// TwinCAT 3 PLC project ProgrammHalle
// ProgramVersion: 3.1.4022.1
// libraries:
//   OSCAT, * (RWTH Aachen University - E.ON Energy Research Center)
//   Tc2_ModbusRTU, * (Beckhoff Automation GmbH)
//   Tc2_Standard, * (Beckhoff Automation GmbH)
//   Tc2_System, * (Beckhoff Automation GmbH)
//   Tc3_BA2_Common, * (Beckhoff Automation GmbH)
//   Tc3_BACnetRev14, * (Beckhoff Automation GmbH)
//   Tc3_BA_Common, * (Beckhoff Automation GmbH)
//   Tc3_IotBase, * (Beckhoff Automation GmbH)
//   Tc3_Module, * (Beckhoff Automation GmbH)
//   TcUnit, * (www.tcunit.org)
// project tree:
//   DUTs/ E_ControlMode.TcDUT, E_PumpControlMode.TcDUT
//   GVLs/ ADS.TcGVL, GVL.TcGVL
//   / PlcTask.TcTTO
//   POUs/Components/ FB_ExhAirModbus.TcPOU, FB_FanBACnet.TcPOU, FB_FanControl.TcPOU, FB_HydMixCir.TcPOU, FB_HydThrotCir.TcPOU, FB_JetNozzle1.TcPOU, FB_JetNozzle2.TcPOU, FB_PumpBACnet.TcPOU, FB_PumpBACnet1.TcPOU, FB_PumpBACnet2.TcPOU, FB_PumpWiloIF.TcPOU, FB_RoomControlUnit.TcPOU, FB_SenTempEL321x.TcPOU, FB_TempSensPt100.TcPOU, FB_TVJModbusMaster.TcPOU, FB_TVRModbusMaster.TcPOU, FB_ValveBACnet.TcPOU, FB_Valve_0_10V.TcPOU, FB_Valve_2_10V.TcPOU, FB_Valve_4_20A.TcPOU, FB_VFCModbus1.TcPOU, FB_VFCModbus2.TcPOU, FB_VVS_JN.TcPOU, FC_CoolingCurve.TcPOU, FC_Current4_20Raw_TO_Percentage.TcPOU, FC_HeatingCurve.TcPOU, FC_MeanOfArray.TcPOU, FC_Percentage_TO_Current4_20Raw.TcPOU, FC_Percentage_TO_Voltage0_10Raw.TcPOU, FC_Percentage_TO_Voltage2_10Raw.TcPOU, FC_Pt100Raw_TO_Temperature.TcPOU, FC_Voltage0_10Raw_TO_Percentage.TcPOU, FC_Voltage2_10Raw_TO_Percentage.TcPOU
//   POUs/EnvTemperature/ FB_AmbientAir.TcPOU
//   POUs/HeatSupplySystem/ FB_HSS.TcPOU, FB_HSSController.TcPOU
//   POUs/Interfaces/ I_Controller.TcIO, I_HydraulicMixingControl.TcIO, I_HydraulicThrottlingControl.TcIO, I_JetNozzle.TcIO, I_Pump.TcIO, I_TemperatureSensor.TcIO, I_Valve.TcIO, I_VolumeFlowController.TcIO
//   POUs/ MAIN.TcPOU
//   POUs/SensorData/ FB_SenDaHydMixCir.TcPOU
//   POUs/Test/Components_Test/ FC_HeatingCurve_Test.TcPOU
//   POUs/Test/HeatSupplySystem_Test/ FB_HSSController_Test.TcPOU
//   POUs/Test/ PRG_TEST.TcPOU

CONFIGURATION ProgrammHalle
    RESOURCE PLC ON TwinCAT3
        TASK PlcTask(INTERVAL := T#10ms, PRIORITY := 20);
        PROGRAM MAIN WITH PlcTask : MAIN;
        PROGRAM PRG_TEST WITH PlcTask : PRG_TEST;
    END_RESOURCE
END_CONFIGURATION

// ---- DUTs/E_ControlMode.TcDUT
{attribute 'qualified_only'}
{attribute 'strict'}
TYPE E_ControlMode :
(
	Off, 				(*0*)
	Init, 				(*1*)
	OperationTest, 		(*2*)
	Auto, 				(*3*)
	Manual,				(*4*)
	ExternalADSControl	(*5*)
);
END_TYPE

// ---- DUTs/E_PumpControlMode.TcDUT
{attribute 'qualified_only'}
{attribute 'strict'}
TYPE E_PumpControlMode :
(
	OFF := 0,					
	CONST_SPEED := 1,				
	CONST_DIFFPRESS := 6,		
	VAR_DIFFPRESS := 7,
	NONE := 99
);
END_TYPE

// ---- GVLs/ADS.TcGVL
{attribute 'qualified_only'}
VAR_GLOBAL
	
	//Modes
	eModeMainControlModeADS	AT %I*	: E_ControlMode := E_ControlMode.Auto; //W
	
	eModeHSSADS			AT %I*	: E_ControlMode := E_ControlMode.Auto; //W
	

	//Ambient air datapoints
	fTempAmbAirADS				AT %Q* 	: REAL;
	fTemperatureAmbientMeanADS 	AT %Q*	: REAL;

	
	//HSS  datapoints
	//Temperature sensor datapoints
	fHSSTempSupPrimADS 	AT %Q*	: REAL;
	fHSSTempRetPrimADS 	AT %Q*	: REAL;
	fHSSTempSupADS 		AT %Q*	: REAL;
	fHSSTempRetADS 		AT %Q*	: REAL;
	//Valve datapoints
	fHSSValveActADS 		AT %Q*	: REAL;
	fHSSValveSetADS 		AT %I*	: REAL;								//W
	//Pump datapoints
	eHSSPumpContModeADS 	AT %I*	: E_PumpControlMode;				//W
	bHSSPumpErrorADS		AT %Q*	: BOOL;
	bHSSPumpOperatingADS 	AT %Q*	: BOOL;
	fHSSPumpPowerADS		AT %Q*	: REAL;
	fHSSPumpPressureADS 	AT %Q*	: REAL;
	bHSSPumpSetOnADS		AT %Q*	: BOOL;
	fHSSPumpSetpointADS	AT %I*	: REAL;								//W
	fHSSPumpSpeedADS		AT %Q*	: REAL;
	fHSSPumpVolFlowADS		AT %Q*	: REAL;
	
	
	
END_VAR

// ---- GVLs/GVL.TcGVL
{attribute 'qualified_only'}
VAR_GLOBAL
	//Ambient air datapoints
	fTempAmbAir		AT %I*	: REAL	:= 10;
	fTemperatureAmbientADS	AT %I*	: REAL	:= -273;
		
	//Temperature sensor datapoints
	fHSSTempSupSet			: REAL;
	fHSSTempSupPrim 		: REAL;
	fHSSTempRetPrim 		: REAL;
	fHSSTempSup 			: REAL;
	fHSSTempRet 			: REAL;
	//Valve datapoints
	bHSSValveError			: BOOL;
	fHSSValveAct 			: REAL;
	fHSSValveSet 			: REAL;
	//Pump datapoints
	eHSSPumpContMode 		: E_PumpControlMode;
	bHSSPumpError			: BOOL;
	bHSSPumpOperating 		: BOOL;
	fHSSPumpPower			: REAL;
	fHSSPumpPressure 		: REAL;
	bHSSPumpSetOn			: BOOL;
	fHSSPumpSetpoint		: REAL;
	fHSSPumpSpeed			: REAL;
	fHSSPumpVolFlow		: REAL;

	
END_VAR

// ---- POUs/Interfaces/I_Controller.TcIO
INTERFACE I_Controller

METHOD Auto
VAR_INPUT
END_VAR
END_METHOD

PROPERTY Error : BOOL
GET
END_GET
SET
END_SET
END_PROPERTY

METHOD Init : BOOL
VAR_INPUT
END_VAR
END_METHOD

METHOD Manual
VAR_INPUT
END_VAR
END_METHOD

PROPERTY Mode : E_ControlMode
GET
END_GET
SET
END_SET
END_PROPERTY

METHOD Off
VAR_INPUT
END_VAR
END_METHOD

METHOD OperationTest : BOOL
VAR_INPUT
END_VAR
END_METHOD

METHOD Run
VAR_INPUT
END_VAR
END_METHOD

END_INTERFACE

// ---- POUs/Interfaces/I_HydraulicMixingControl.TcIO
INTERFACE I_HydraulicMixingControl EXTENDS I_Controller

PROPERTY PumpMode : E_PumpControlMode
GET
END_GET
SET
END_SET
END_PROPERTY

PROPERTY PumpSet : REAL
GET
END_GET
SET
END_SET
END_PROPERTY

PROPERTY TemperatureSupAct : REAL
GET
END_GET
SET
END_SET
END_PROPERTY

PROPERTY TemperatureSupSet : REAL
GET
END_GET
SET
END_SET
END_PROPERTY

PROPERTY ValveSet : REAL
GET
END_GET
SET
END_SET
END_PROPERTY

END_INTERFACE

// ---- POUs/Interfaces/I_HydraulicThrottlingControl.TcIO
INTERFACE I_HydraulicThrottlingControl EXTENDS I_Controller

PROPERTY PumpMode : E_PumpControlMode
GET
END_GET
SET
END_SET
END_PROPERTY

PROPERTY PumpSet : REAL
GET
END_GET
SET
END_SET
END_PROPERTY

PROPERTY TemperatureSupAct : REAL
GET
END_GET
SET
END_SET
END_PROPERTY

PROPERTY TemperatureSupSet : REAL
GET
END_GET
SET
END_SET
END_PROPERTY

PROPERTY ValveSet : REAL
GET
END_GET
SET
END_SET
END_PROPERTY

END_INTERFACE

// ---- POUs/Interfaces/I_JetNozzle.TcIO
INTERFACE I_JetNozzle

PROPERTY AngleActual : REAL
GET
END_GET
SET
END_SET
END_PROPERTY

PROPERTY AngleSetpoint : REAL
GET
END_GET
SET
END_SET
END_PROPERTY

PROPERTY Error : BOOL
GET
END_GET
SET
END_SET
END_PROPERTY

METHOD Run
VAR_INPUT
END_VAR
END_METHOD

END_INTERFACE

// ---- POUs/Interfaces/I_Pump.TcIO
INTERFACE I_Pump

PROPERTY ControlMode : E_PumpControlMode
GET
END_GET
SET
END_SET
END_PROPERTY

PROPERTY Error : BOOL
GET
END_GET
SET
END_SET
END_PROPERTY

PROPERTY Operating : BOOL
GET
END_GET
SET
END_SET
END_PROPERTY

PROPERTY PowerRating : REAL
GET
END_GET
SET
END_SET
END_PROPERTY

PROPERTY Pressure : REAL
GET
END_GET
SET
END_SET
END_PROPERTY

METHOD Run
VAR_INPUT
END_VAR
END_METHOD

PROPERTY SetOn : BOOL
GET
END_GET
SET
END_SET
END_PROPERTY

PROPERTY Setpoint : REAL
GET
END_GET
SET
END_SET
END_PROPERTY

PROPERTY Speed : REAL
GET
END_GET
SET
END_SET
END_PROPERTY

PROPERTY VolumeFlow : REAL
GET
END_GET
SET
END_SET
END_PROPERTY

END_INTERFACE

// ---- POUs/Interfaces/I_TemperatureSensor.TcIO
INTERFACE I_TemperatureSensor

METHOD Run
VAR_INPUT
END_VAR
END_METHOD

PROPERTY Temperature : REAL
GET
END_GET
SET
END_SET
END_PROPERTY

END_INTERFACE

// ---- POUs/Interfaces/I_Valve.TcIO
INTERFACE I_Valve

PROPERTY Error : BOOL
GET
END_GET
SET
END_SET
END_PROPERTY

PROPERTY OpeningActual : REAL
GET
END_GET
SET
END_SET
END_PROPERTY

PROPERTY OpeningSetpoint : REAL
GET
END_GET
SET
END_SET
END_PROPERTY

METHOD Run
VAR_INPUT
END_VAR
END_METHOD

END_INTERFACE

// ---- POUs/Interfaces/I_VolumeFlowController.TcIO
INTERFACE I_VolumeFlowController

PROPERTY Error : BOOL
GET
END_GET
SET
END_SET
END_PROPERTY

METHOD Run : BOOL
VAR_INPUT
END_VAR
END_METHOD

PROPERTY VolumeFlowActual : REAL
GET
END_GET
SET
END_SET
END_PROPERTY

PROPERTY VolumeFlowSetpoint : REAL
GET
END_GET
SET
END_SET
END_PROPERTY

END_INTERFACE

// ---- POUs/MAIN.TcPOU
PROGRAM MAIN
VAR
	//Control mode
	eMode : E_ControlMode := E_ControlMode.Auto;
	
	// Heat supply circle
	fbHSS		: FB_HSS;

	//simulated sensor data
	fbHSSSenDa	: FB_SenDaHydMixCir;
	//simulated enviromental temperature
	fbAmbientAir : FB_AmbientAir;		
								 
END_VAR

//Check main control mode
eMode := ADS.eModeMainControlModeADS;
//Set control modes
IF eMode = E_ControlMode.ExternalADSControl THEN		
	fbHSS.Mode 	:= ADS.eModeHSSADS;	
ELSE	
	fbHSS.Mode 	:= eMode;
END_IF

//Simulated the sensor tmeprature and enviromental temperature
 
fbHSSSenDa.Run();
fbAmbientAir.Run();

//Raw temperature input 
fbHSS.TempSupPrim := fbHSSSenDa.fTempSupPrimAct;
fbHSS.TempRetPrim := fbHSSSenDa.fTempRetPrimAct;
fbHSS.TempRet := fbHSSSenDa.fTempRetAct;
fbHSS.TempSup := fbHSSSenDa.fTempSupAct;
//Valve input
fbHSS.Valve := fbHSSSenDa.fHSSValveAct;


//Execute Routine 
fbHSS.Run();

END_PROGRAM

// ---- POUs/HeatSupplySystem/FB_HSS.TcPOU
FUNCTION_BLOCK FB_HSS
VAR_INPUT
END_VAR
VAR_OUTPUT
END_VAR
VAR
	//Properties
	bError 			: BOOL 				:= FALSE;
	eMode 			: E_ControlMode 	:= E_ControlMode.Off;	
	//Components
	//Valve
	fbValve 		:	FB_Valve_4_20A;
	//Pump with BACnet client
	fbPump 			:	FB_PumpBACnet2 :=(fbClient:=(nDeviceInstance:=16));
	//Temperature sensors
	fbTempSupPrim 	: 	FB_TempSensPt100;
	fbTempRetPrim 	: 	FB_TempSensPt100;
	fbTempSup 		: 	FB_TempSensPt100;
	fbTempRet 		: 	FB_TempSensPt100;
	//Controller
	fbControl 		: 	FB_HSSController;
	//Hydraulic circuit
	fbHydCir		: FB_HydMixCir := (	iPump 			:= fbPump,
										iValve			:= fbValve,
										iTempSupPrim 	:= fbTempSupPrim,
										iTempRetPrim 	:= fbTempRetPrim,
										iTempSup 		:= fbTempSup,
										iTempRet 		:= fbTempRet,
										iControl 		:= fbControl);
END_VAR

PROPERTY PUBLIC Error : BOOL
GET
Error := THIS^.bError;
END_GET
SET
THIS^.bError := Error;
END_SET
END_PROPERTY

PROPERTY PUBLIC Mode : E_ControlMode
GET
Mode := THIS^.eMode;
END_GET
SET
THIS^.eMode := Mode;
END_SET
END_PROPERTY

METHOD Run
VAR_INPUT
END_VAR
//Execute hydraulic circuit with its control routine
fbHydCir.Mode := eMode;
fbHydCir.Run();

//Write values to GVL
//Temperature datapoints
GVL.fHSSTempSupPrim 	:= fbTempSupPrim.Temperature;
GVL.fHSSTempRetPrim 	:= fbTempRetPrim.Temperature;
GVL.fHSSTempSup 		:= fbTempSup.Temperature;
GVL.fHSSTempRet 		:= fbTempRet.Temperature;
//ADS
ADS.fHSSTempSupPrimADS 	:= fbTempSupPrim.Temperature;
ADS.fHSSTempRetPrimADS 	:= fbTempRetPrim.Temperature;
ADS.fHSSTempSupADS 		:= fbTempSup.Temperature;
ADS.fHSSTempRetADS 		:= fbTempRet.Temperature;


//Valve datapoints
GVL.bHSSValveError 	:= fbValve.Error;
GVL.fHSSValveSet 		:= fbValve.OpeningSetpoint;
GVL.fHSSValveAct 		:= fbValve.OpeningActual;
//ADS
ADS.fHSSValveActADS 	:= fbValve.OpeningActual;


//Pump datapoints
GVL.eHSSPumpContMode	:= fbPump.ControlMode;
GVL.bHSSPumpError 		:= fbPump.Error;
GVL.bHSSPumpOperating	:= fbPump.Operating;
GVL.fHSSPumpPower		:= fbPump.PowerRating;
GVL.fHSSPumpPressure 	:= fbPump.Pressure;
GVL.bHSSPumpSetOn		:= fbPump.SetOn;
GVL.fHSSPumpSetpoint	:= fbPump.Setpoint;
GVL.fHSSPumpSpeed		:= fbPump.Speed;
GVL.fHSSPumpVolFlow	:= fbPump.VolumeFlow;
//ADS
ADS.bHSSPumpErrorADS 		:= fbPump.Error;
ADS.bHSSPumpOperatingADS	:= fbPump.Operating;
ADS.fHSSPumpPowerADS		:= fbPump.PowerRating;
ADS.fHSSPumpPressureADS 	:= fbPump.Pressure;
ADS.bHSSPumpSetOnADS		:= fbPump.SetOn;
ADS.fHSSPumpSpeedADS		:= fbPump.Speed;
ADS.fHSSPumpVolFlowADS		:= fbPump.VolumeFlow;
END_METHOD

PROPERTY PUBLIC TempRet : REAL
GET
TempRet:= THIS^.fbTempRet.TempRaw;
END_GET
SET
THIS^.fbTempRet.TempRaw := TempRet;
END_SET
END_PROPERTY

PROPERTY PUBLIC TempRetPrim : REAL
GET
TempRetPrim:= THIS^.fbTempRetPrim.TempRaw;
END_GET
SET
THIS^.fbTempRetPrim.TempRaw := TempRetPrim;
END_SET
END_PROPERTY

PROPERTY PUBLIC TempSup : REAL
GET
TempSup := THIS^.fbTempSup.TempRaw;
END_GET
SET
THIS^.fbTempSup.TempRaw := TempSup;
END_SET
END_PROPERTY

PROPERTY PUBLIC TempSupPrim : REAL
GET
TempSupPrim := THIS^.fbTempSupPrim.TempRaw;
END_GET
SET
THIS^.fbTempSupPrim.TempRaw := TempSupPrim;
END_SET
END_PROPERTY

PROPERTY PUBLIC Valve : REAL
GET
Valve := THIS^.fbValve.nOpeningAct;
END_GET
SET
THIS^.fbValve.nOpeningAct := Valve;
END_SET
END_PROPERTY

END_FUNCTION_BLOCK

// ---- POUs/Components/FB_Valve_4_20A.TcPOU
FUNCTION_BLOCK FB_Valve_4_20A IMPLEMENTS I_Valve
VAR_INPUT
	nOpeningAct AT %I* : REAL;
END_VAR
VAR_OUTPUT
END_VAR
VAR
		//Properties
	bError : BOOL := FALSE;
	fOpeningActual : REAL;
	fOpeningSetpoint : REAL := 0;
	//Raw values
	nOpeningSet AT %Q* : INT;
	//nOpeningAct AT %I* : INT;
END_VAR

PROPERTY Error : BOOL
GET
Error := THIS^.bError;
END_GET
SET
THIS^.bError := Error;
END_SET
END_PROPERTY

PROPERTY OpeningActual : REAL
GET
OpeningActual := THIS^.fOpeningActual;
END_GET
SET
THIS^.fOpeningActual := OpeningActual;
END_SET
END_PROPERTY

PROPERTY OpeningSetpoint : REAL
GET
OpeningSetpoint := THIS^.fOpeningSetpoint;
END_GET
SET
THIS^.fOpeningSetpoint := OpeningSetpoint;
END_SET
END_PROPERTY

METHOD Run
VAR_INPUT
END_VAR
//Read feedback for opening position
fOpeningActual := FC_Current4_20Raw_TO_Percentage(nOpeningAct);

//Write setpoint for opening position
nOpeningSet := FC_Percentage_TO_Current4_20Raw(fOpeningSetpoint);
END_METHOD

END_FUNCTION_BLOCK

// ---- POUs/Components/FC_Current4_20Raw_TO_Percentage.TcPOU
FUNCTION FC_Current4_20Raw_TO_Percentage : REAL
VAR_INPUT
	i : REAL;
END_VAR
VAR
	f : REAL;
	nIntMax : REAL := 32767;
	nIntMin : REAL := 6553;
END_VAR

FC_Current4_20Raw_TO_Percentage := 100*(i-nIntMin)/(nIntMax-nIntMin);

END_FUNCTION

// ---- POUs/Components/FC_Percentage_TO_Current4_20Raw.TcPOU
FUNCTION FC_Percentage_TO_Current4_20Raw : INT
VAR_INPUT
	f : REAL;
END_VAR
VAR
	nIntMax : INT := 32767;
	nIntMin : INT := 6553;
END_VAR

FC_Percentage_TO_Current4_20Raw := REAL_TO_INT(nIntMin + (f/100)*(nIntMax-nIntMin));

END_FUNCTION

// ---- POUs/Components/FB_PumpBACnet2.TcPOU
FUNCTION_BLOCK FB_PumpBACnet2 IMPLEMENTS I_Pump
VAR_INPUT CONSTANT
	fbClient : FB_BACnet_Client;
END_VAR
VAR_OUTPUT
END_VAR
VAR
	//Properties
	eControlMode : E_PumpControlMode := E_PumpControlMode.OFF;
	bError : BOOL;
	bOperating : BOOL;
	fPowerRating : REAL;
	fPressure : REAL;
	bSetOn : BOOL := FALSE;
	fSetpoint : REAL := 0;
	fSpeed : REAL;
	fVolumeFlow : REAL;	

	//BACnet parameters
	nPriority : BYTE := 12;
	
	//BACnet Mapping
	ContModeBAC		:	FB_BACnetRM_MO := (Client := fbClient, nObjectInstance :=0);		//Pump Control mode (speed, var/const pressure)
	ErrorBAC		:	FB_BACnetRM_BI := (Client := fbClient, nObjectInstance :=13);		//Error
	OperatingBAC	:	FB_BACnetRM_BI := (Client := fbClient, nObjectInstance :=10);		//Operation active/inactive
	PowerRatingBAC	:	FB_BACnetRM_AI := (Client := fbClient, nObjectInstance :=4);		//Current power
	PressureBAC		:	FB_BACnetRM_AI := (Client := fbClient, nObjectInstance :=3);		//Estimated pressure difference
	SetpointBAC		:	FB_BACnetRM_AO := (Client := fbClient, nObjectInstance :=0);		//Setpoint
	SetOnBAC		:	FB_BACnetRM_BO := (Client := fbClient, nObjectInstance :=0);		//Turn on/off
	SpeedBAC		:	FB_BACnetRM_AI := (Client := fbClient, nObjectInstance :=1);		//Estimated speed
	VolumeFlowBAC	:	FB_BACnetRM_AI := (Client := fbClient, nObjectInstance :=2);		//Estimated volume flow

END_VAR

PROPERTY ControlMode : E_PumpControlMode
GET
ControlMode := THIS^.eControlMode;
END_GET
SET
THIS^.eControlMode := ControlMode;
END_SET
END_PROPERTY

PROPERTY Error : BOOL
GET
Error := THIS^.bError;
END_GET
SET
THIS^.bError := Error;
END_SET
END_PROPERTY

PROPERTY Operating : BOOL
GET
Operating := THIS^.bOperating;
END_GET
SET
THIS^.bOperating := Operating;
END_SET
END_PROPERTY

PROPERTY PowerRating : REAL
GET
PowerRating := THIS^.fPowerRating;
END_GET
SET
THIS^.fPowerRating := PowerRating;
END_SET
END_PROPERTY

PROPERTY Pressure : REAL
GET
Pressure := THIS^.fPressure;
END_GET
SET
THIS^.fPressure := Pressure;
END_SET
END_PROPERTY

METHOD Run
//Run BACnet Client
(*fbClient();

//Read BACnet values
ErrorBAC(bPresentValue=>bError);
OperatingBAC(bPresentValue=>bOperating);
PowerRatingBAC(fPresentValue=>fPowerRating);
PressureBAC(fPresentValue=>fPressure);
SpeedBAC(fPresentValue=>fSpeed);
VolumeFlowBAC(fPresentValue=>fVolumeFlow);

//Write BACnet values
//Set pump values depending on defined ControlMode
IF eControlMode = E_PumpControlMode.OFF THEN
	//Set pump to off
	SetOnBAC(bPv:=FALSE,bEnablePv:=TRUE,ePriority:=nPriority);
	ContModeBAC(nPv:=eControlMode,bEnablePv:=TRUE,ePriority:=nPriority);
	SetpointBAC(fPv:=0,bEnablePv:=TRUE,ePriority:=nPriority);
ELSIF eControlMode = E_PumpControlMode.NONE THEN
	//Release
	SetOnBAC(bNullPv:=TRUE,ePriority:=nPriority); 	//Clear entry
	ContModeBAC(bNullPv:=TRUE,ePriority:=nPriority); //Clear entry
	SetpointBAC(bNullPv:=TRUE,ePriority:=nPriority); //Clear entry
ELSE
	//Set pump to on and set setpoint
	SetOnBAC(bPV:=TRUE,bEnablePv:=TRUE,ePriority:=nPriority);
	ContModeBAC(nPV:=eControlMode,bEnablePv:=TRUE,ePriority:=nPriority);
	SetpointBAC(fPV:=fSetpoint,bEnablePv:=TRUE,ePriority:=nPriority);
END_IF

*)
END_METHOD

PROPERTY SetOn : BOOL
GET
SetOn := THIS^.bSetOn;
END_GET
SET
THIS^.bSetOn := SetOn;
END_SET
END_PROPERTY

PROPERTY Setpoint : REAL
GET
Setpoint := THIS^.fSetpoint;
END_GET
SET
THIS^.fSetpoint := Setpoint;
END_SET
END_PROPERTY

PROPERTY Speed : REAL
GET
Speed := THIS^.fSpeed;
END_GET
SET
THIS^.fSpeed := Speed;
END_SET
END_PROPERTY

PROPERTY VolumeFlow : REAL
GET
VolumeFlow := THIS^.fVolumeFlow;
END_GET
SET
THIS^.fVolumeFlow := VolumeFlow;
END_SET
END_PROPERTY

END_FUNCTION_BLOCK

// ---- POUs/Components/FB_TempSensPt100.TcPOU
FUNCTION_BLOCK FB_TempSensPt100 IMPLEMENTS I_TemperatureSensor
VAR_INPUT
	TempRaw AT %I* : REAL;
END_VAR
VAR_OUTPUT
END_VAR
VAR
	//Properties
	fTemperature : REAL;
	//Raw value
	
END_VAR

METHOD Run
//Read temperature
fTemperature :=  FC_Pt100Raw_TO_Temperature(TempRaw);
END_METHOD

PROPERTY Temperature : REAL
GET
Temperature := THIS^.fTemperature;
END_GET
SET
THIS^.fTemperature := Temperature;
END_SET
END_PROPERTY

END_FUNCTION_BLOCK

// ---- POUs/Components/FC_Pt100Raw_TO_Temperature.TcPOU
FUNCTION FC_Pt100Raw_TO_Temperature : REAL
VAR_INPUT
	i : REAL;
END_VAR
VAR
	ConvFac : REAL := 10;
END_VAR

FC_Pt100Raw_TO_Temperature := (i)/ConvFac;

END_FUNCTION

// ---- POUs/HeatSupplySystem/FB_HSSController.TcPOU
FUNCTION_BLOCK FB_HSSController IMPLEMENTS I_HydraulicMixingControl
VAR_INPUT
END_VAR
VAR_OUTPUT
END_VAR
VAR
	//Properties
	bError 			: BOOL 				:= FALSE;
	eMode 			: E_ControlMode 	:= E_ControlMode.Off;
	ePumpMode 		: E_PumpControlMode := E_PumpControlMode.OFF;
	fPumpSet 		: REAL 				:= 0;
	fTemperatureAct : REAL              := 18;
	fTemperatureSet : REAL				:= 45;
	fValveSet 		: REAL 				:= 0;
	
	//PID
	fbPID : FB_PID; //Set PID parameters (Kp, Ti, ...) in Auto method
	
	//Manual mode
	eManualPumpMode	: E_PumpControlMode := E_PumpControlMode.NONE;
	fManualPumpSet	: REAL 				:= fPumpSet;
	fManualValveSet : REAL 				:= fValveSet;
	
END_VAR

METHOD Auto
VAR
	//PID params
	Kp		:	REAL	:=	1.4;	//Proportional gain
	Ti		:	REAL	:=	80;		//Integral time
	Td		:	REAL	:=	0;		//Derivative time
	LimLow	:	REAL	:=	0;		//Low limit of output
	LimHigh	:	REAL	:=	100;	//High limit of output
	bReverseActing	:	BOOL := FALSE;
	
	//Heating Curve
	fSlope	: 	REAL	:= 	-1.0;
	fOffset	: 	REAL	:= 	45.0;
END_VAR
//TROX controls heating power via throttle circuit
//Calculate supply water set temperature from heating curve, 45 °C at 0 °C ambient temperature

fTemperatureSet := FC_HeatingCurve(	fTempAmb := GVL.fTempAmbAir,
									fSlope := fSlope,
									fOffset := fOffset);

//PID control for valve
fbPID(
	xSet:= fTemperatureSet, 
	xAct:= fTemperatureAct, 
	Kp:= Kp, 
	Ti:= Ti, 
	Td:= Td, 
	LimLow:= LimLow, 
	LimHigh:= LimHigh, 
	bReverseActing:= bReverseActing, 
	RST:= FALSE, 
	Y=> fValveSet
	);

//Pump setpoint just constant for now
fPumpSet 	:= 60; //60 % of nominal power
ePumpMode 	:= E_PumpControlMode.CONST_DIFFPRESS;
END_METHOD

PROPERTY Error : BOOL
GET
Error := THIS^.bError;
END_GET
SET
THIS^.bError := Error;
END_SET
END_PROPERTY

METHOD ExternalADSControl
VAR_INPUT
END_VAR
//Set Valve position according to ADS command
fValveSet := ADS.fHSSValveSetADS;

//Set pump operation and set point to ADS command
fPumpSet 	:= ADS.fHSSPumpSetpointADS; // % of nominal power
ePumpMode 	:= ADS.eHSSPumpContModeADS;
END_METHOD

{warning 'add method implementation '}
METHOD Init : BOOL
END_METHOD

METHOD Manual
ePumpMode 	:= eManualPumpMode;
fPumpSet 	:= fManualPumpSet;
fValveSet 	:= fManualValveSet;
END_METHOD

PROPERTY Mode : E_ControlMode
GET
Mode := THIS^.eMode;
END_GET
SET
THIS^.eMode := Mode;
END_SET
END_PROPERTY

METHOD Off
fPumpSet	:=	0;
ePumpMode	:=	E_PumpControlMode.OFF;
fValveSet 	:=	0;
END_METHOD

{warning 'add method implementation '}
METHOD OperationTest : BOOL
END_METHOD

PROPERTY PumpMode : E_PumpControlMode
GET
PumpMode := THIS^.ePumpMode;
END_GET
SET
THIS^.ePumpMode := PumpMode;
END_SET
END_PROPERTY

PROPERTY PumpSet : REAL
GET
PumpSet := THIS^.fPumpSet;
END_GET
SET
THIS^.fPumpSet := PumpSet;
END_SET
END_PROPERTY

METHOD Run
//Run control routine according to mode set
CASE eMode OF
	E_ControlMode.Off:		   			Off();
	E_ControlMode.Init:		   			Init();
	E_ControlMode.OperationTest:	    OperationTest();
	E_ControlMode.Auto:   				Auto();
	E_ControlMode.Manual:				Manual();
	E_ControlMode.ExternalADSControl:	ExternalADSControl();
END_CASE

//Write temperature supply setpoint to GVL
GVL.fHSSTempSupSet := THIS^.TemperatureSupSet;
END_METHOD

PROPERTY TemperatureSupAct : REAL
GET
TemperatureSupAct := THIS^.fTemperatureAct;
END_GET
SET
THIS^.fTemperatureAct := TemperatureSupAct;
END_SET
END_PROPERTY

PROPERTY TemperatureSupSet : REAL
GET
TemperatureSupSet := THIS^.fTemperatureSet;
END_GET
SET
THIS^.fTemperatureSet := TemperatureSupSet;
END_SET
END_PROPERTY

PROPERTY ValveSet : REAL
GET
ValveSet := THIS^.fValveSet;
END_GET
SET
THIS^.fValveSet := ValveSet;
END_SET
END_PROPERTY

END_FUNCTION_BLOCK

// ---- POUs/Components/FC_HeatingCurve.TcPOU
FUNCTION FC_HeatingCurve : REAL
VAR_INPUT
	fTempAmb 	: REAL; 		//Ambient temperature
	fSlope 		: REAL := -1; 	//Slope of heatcurve
	fOffset 	: REAL := 35;	//In °C; off set at T_amb=0°C
END_VAR
VAR
END_VAR
VAR CONSTANT 
END_VAR

FC_HeatingCurve:= fSlope * fTempAmb + fOffset;

END_FUNCTION

// ---- POUs/Components/FB_HydMixCir.TcPOU
FUNCTION_BLOCK FB_HydMixCir
VAR_INPUT
	//Pump
	iPump			:	I_Pump;
	//Valve
	iValve			:	I_Valve;
	//Temperatures
	iTempSupPrim	:	I_TemperatureSensor;
	iTempRetPrim	:	I_TemperatureSensor;
	iTempSup		:	I_TemperatureSensor;
	iTempRet		:	I_TemperatureSensor;
	//Controller
	iControl		:	I_HydraulicMixingControl;
END_VAR
VAR_OUTPUT
END_VAR
VAR
	eMode : E_ControlMode := E_ControlMode.Off;
END_VAR

PROPERTY Mode : E_ControlMode
GET
Mode := THIS^.eMode;
END_GET
SET
THIS^.eMode := Mode;
END_SET
END_PROPERTY

METHOD Run
VAR_INPUT
END_VAR
//Update temperatures
iTempSupPrim.Run();
iTempRetPrim.Run();
iTempSup.Run();
iTempRet.Run();

//Run components
iPump.Run();
iValve.Run();

//Run controller
iControl.Mode := eMode;
iControl.TemperatureSupAct := iTempSup.Temperature;
iControl.Run();

//Pump set properties
IF eMode = E_ControlMode.Off THEN
	iPump.SetOn := FALSE;
ELSE
	iPump.SetOn := TRUE;
END_IF
iPump.ControlMode := iControl.PumpMode;
iPump.Setpoint := iControl.PumpSet;

//Valve set properties
iValve.OpeningSetpoint := iControl.ValveSet;
END_METHOD

END_FUNCTION_BLOCK

// ---- POUs/SensorData/FB_SenDaHydMixCir.TcPOU
FUNCTION_BLOCK FB_SenDaHydMixCir
VAR_INPUT
END_VAR
VAR_OUTPUT
END_VAR
VAR
	ftemp_sensor : OSCAT.GEN_RMP:= ( PT := T#10S,
								     AM := 150,
								     OS := 80,
								     DL:= 0);
	fvalve_act : OSCAT.GEN_RMP := ( PT := T#100S,
								     AM := 52428,
								     OS := -19661,
								     DL:= 0);
// variable for valve, pump
	fTempSupPrimAct: REAL;
	fTempRetPrimAct: REAL;
	fTempSupAct: REAL;
	fTempRetAct: REAL;
	
	fHSSValveAct: REAL;
	
	
END_VAR

METHOD Run
VAR_INPUT
END_VAR

ftemp_sensor();
fTempSupPrimAct := ftemp_sensor.OUT ;
fTempRetPrimAct := ftemp_sensor.OUT ;
fTempSupAct := ftemp_sensor.OUT;
fTempRetAct := ftemp_sensor.OUT ;

fvalve_act();
fHSSValveAct := fvalve_act.OUT;
END_METHOD

END_FUNCTION_BLOCK

// ---- POUs/EnvTemperature/FB_AmbientAir.TcPOU
FUNCTION_BLOCK FB_AmbientAir 
VAR_INPUT
END_VAR
VAR_OUTPUT
END_VAR
VAR
	ftemp_sin: OSCAT.GEN_SIN:= ( PT := T#10S,
								     AM := 7,
								     OS := 12,
								     DL:= 0); 
END_VAR

METHOD Run 
VAR_INPUT
END_VAR
ftemp_sin();
GVL.fTempAmbAir := ftemp_sin.Out;
END_METHOD

END_FUNCTION_BLOCK

// ---- POUs/Test/PRG_TEST.TcPOU
PROGRAM PRG_TEST
VAR
	HeatingCurve_Test : FC_HeatingCurve_Test;							 
END_VAR

TcUnit.RUN();

END_PROGRAM

// ---- POUs/Test/Components_Test/FC_HeatingCurve_Test.TcPOU
FUNCTION_BLOCK FC_HeatingCurve_Test EXTENDS TcUnit.FB_TestSuite
VAR
END_VAR

NegativeTAmb();
TAmbZero();
HeatingCurveZero();
NegativeHeatingCurve();

METHOD FB_init : BOOL
VAR_INPUT
    bInitRetains : BOOL; // if TRUE, the retain variables are initialized (warm start / cold start)
    bInCopyCode : BOOL;  // if TRUE, the instance afterwards gets moved into the copy code (online change)
END_VAR
END_METHOD

METHOD HeatingCurveZero
VAR
	HeatingCurve: FC_HeatingCurve;
	ExpectedValue : REAL := 0;
	fSlope: REAL;
	fOffset: REAL;

END_VAR
TEST('HeatingCurveZero');
 
HeatingCurve(fTempAmb := 35, fSlope, fOffset);
 
AssertEquals(Expected := ExpectedValue,
             Actual := HeatingCurve,
             Message := 'The calculation is not correct');
 
TEST_FINISHED();
END_METHOD

METHOD NegativeHeatingCurve
VAR
	HeatingCurve: FC_HeatingCurve;
	ExpectedValue : REAL := -1;
	fSlope: REAL;
	fOffset: REAL;
END_VAR
TEST('NegativeHeatingCurve');
 
HeatingCurve(fTempAmb := 36, fSlope, fOffset);
 
AssertEquals(Expected := ExpectedValue,
             Actual := HeatingCurve,
             Message := 'The calculation is not correct');
 
TEST_FINISHED();
END_METHOD

METHOD NegativeTAmb
VAR
	HeatingCurve: FC_HeatingCurve;
	ExpectedValue : REAL := 40;
	fSlope: REAL;
	fOffset: REAL;
END_VAR
TEST('NegativeTAmb');
 
HeatingCurve(fTempAmb := -5, fSlope, fOffset);
 
AssertEquals(Expected := ExpectedValue,
             Actual := HeatingCurve,
             Message := 'The calculation is not correct');
 
TEST_FINISHED();
END_METHOD

METHOD TAmbZero
VAR
	HeatingCurve: FC_HeatingCurve;
	ExpectedValue : REAL := 35;
	fSlope: REAL;
	fOffset: REAL;

END_VAR
TEST('TAmbZero');
 
HeatingCurve(fTempAmb := 0, fSlope, fOffset);
 
AssertEquals(Expected := ExpectedValue,
             Actual := HeatingCurve,
             Message := 'The calculation is not correct');
 
TEST_FINISHED();
END_METHOD

END_FUNCTION_BLOCK

// ---- POUs/Components/FB_ExhAirModbus.TcPOU
FUNCTION_BLOCK FB_ExhAirModbus
VAR_INPUT
	nSet	:	WORD;	//Setpoint in hundreds of a percent
END_VAR
VAR_OUTPUT
	nAct	:	Array[11..12] of WORD;	//Actual volume flow in m^3/h
END_VAR
VAR
	Step	:	INT		:=	1;
	ModAdr	:	BYTE	:=	11;
	
	nZwang	:	WORD;
	bZwang	:	BOOL	:=	FALSE;
	
	fbModK6		:	ModbusRtuMaster_KL6x22B;
	bModErr		:	BOOL;
	ErrID		:	MODBUS_ERRORS;
END_VAR

CASE Step OF
	
	1:	//start writing setpoint to nozzle
		IF nSet = 65535 THEN
			Step	:=	20;	//Control override
			bZwang	:=	TRUE;
		ELSE
			IF bZwang THEN
				Step :=	30;
			ELSE
				fbModK6.WriteSingleRegister(
						UnitID		:=	ModAdr,	//Modbus address of slave
						MBAddr		:=	0,	//Register address
						Quantity	:=	1,	//Number of registers to be written
						pMemoryAddr	:=	ADR(nSet),		//Pointer to write data
						cbLength	:=	SIZEOF(nSet),	//Size of write data
						Timeout		:=	T#5S,			//Time to wait for the slave to respond
						Execute		:=	TRUE
					);
					Step	:=	2;
			END_IF
		END_IF
		
	2:	//finish writing process
		fbModK6.WriteSingleRegister(Execute:=FALSE, Error=>bModErr, ErrorID=>ErrID);
		IF NOT fbModK6.BUSY THEN
			Step	:=	3;	//go to next step when writing process has finished
		END_IF
		IF fbModK6.Error THEN
			Step	:=	99;
		END_IF
		
	3:	//start reading volume flow
		fbModK6.ReadRegs(
			UnitID		:=	ModAdr,	//Modbus address of slave
			MBAddr		:=	7,	//Register address
			Quantity	:=	1,	//Number of registers to be read
			pMemoryAddr	:=	ADR(nAct[ModAdr]),		//Pointer to read data
			cbLength	:=	SIZEOF(nAct[ModAdr]),	//Size of read data
			Timeout		:=	T#5S,			//Time to wait for the slave to respond
			Execute		:=	TRUE
		);
		Step	:=	4;
		
	4:	//finish reading process
		fbModK6.ReadRegs(Execute:=FALSE, Error=>bModErr, ErrorID=>ErrID);
		IF NOT fbModK6.BUSY THEN
			Step	:=	5;	//go to next step when reading process has finished
		END_IF
		IF fbModK6.Error THEN
			Step	:=	99;
		END_IF
		
	5:	//go to next nozzle or finish operation
		ModAdr	:=	ModAdr+1;
		IF ModAdr <= 12 THEN
			Step	:=	1;	//start process for other actuator
		ELSE
			Step	:=	6;
		END_IF
		
	6:	//prepare next operation
		ModAdr	:=	11;
		Step	:=	1;
		
	20: //Activate control override for actuator 1
		nZwang	:=	2;
		fbModK6.WriteSingleRegister(
			UnitID		:=	11,	//Modbus address of slave
			MBAddr		:=	1,	//Regster address
			Quantity	:=	1,	//Number of registers to be written
			pMemoryAddr	:=	ADR(nZwang),		//Pointer to write data
			cbLength	:=	SIZEOF(nZwang),	//Size of write data
			Timeout		:=	T#5S,				//Time to wait for the slave to respond
			Execute		:=	TRUE
		);
		Step	:=	21;
	
	21:	//finish writing process
		fbModK6.WriteSingleRegister(Execute:=FALSE, Error=>bModErr, ErrorID=>ErrID);
		IF NOT fbModK6.BUSY THEN
			Step	:=	22;	//go to next step when writing process has finished
		END_IF
		IF fbModK6.Error THEN
			Step	:=	99;
		END_IF
		
	22: //Activate control override for actuator 2		
		nZwang	:=	2;
		fbModK6.WriteSingleRegister(
			UnitID		:=	12,	//Modbus address of slave
			MBAddr		:=	1,	//Regster address
			Quantity	:=	1,	//Number of registers to be written
			pMemoryAddr	:=	ADR(nZwang),		//Pointer to write data
			cbLength	:=	SIZEOF(nZwang),	//Size of write data
			Timeout		:=	T#5S,				//Time to wait for the slave to respond
			Execute		:=	TRUE
		);
		Step	:=	23;
	
	23:	//finish writing process
		fbModK6.WriteSingleRegister(Execute:=FALSE, Error=>bModErr, ErrorID=>ErrID);
		IF NOT fbModK6.BUSY THEN
			Step	:=	3;	//go to next step when writing process has finished
		END_IF
		IF fbModK6.Error THEN
			Step	:=	99;
		END_IF
		
	30: //End control override for actuator 1
		nZwang	:=	0;
		fbModK6.WriteSingleRegister(
			UnitID		:=	11,	//Modbus address of slave
			MBAddr		:=	1,	//Register address
			Quantity	:=	1,	//Number of registers to be written
			pMemoryAddr	:=	ADR(nZwang),		//Pointer to write data
			cbLength	:=	SIZEOF(nZwang),	//Size of write data
			Timeout		:=	T#5S,				//Time to wait for the slave to respond
			Execute		:=	TRUE
		);
		Step	:=	31;
	
	31:	//finish writing process
		fbModK6.WriteSingleRegister(Execute:=FALSE, Error=>bModErr, ErrorID=>ErrID);
		IF NOT fbModK6.BUSY THEN
			bZwang	:=	FALSE;
			Step	:=	32;
		END_IF
		IF fbModK6.Error THEN
			Step	:=	99;
		END_IF
		
	32: //End control override for actuator 2
		nZwang	:=	0;
		fbModK6.WriteSingleRegister(
			UnitID		:=	12,	//Modbus address of slave
			MBAddr		:=	1,	//Register address
			Quantity	:=	1,	//Number of registers to be written
			pMemoryAddr	:=	ADR(nZwang),		//Pointer to write data
			cbLength	:=	SIZEOF(nZwang),	//Size of write data
			Timeout		:=	T#5S,				//Time to wait for the slave to respond
			Execute		:=	TRUE
		);
		Step	:=	33;
	
	33:	//finish writing process
		fbModK6.WriteSingleRegister(Execute:=FALSE, Error=>bModErr, ErrorID=>ErrID);
		IF NOT fbModK6.BUSY THEN
			bZwang	:=	FALSE;
			Step	:=	1;	//start normal writing process
		END_IF
		IF fbModK6.Error THEN
			Step	:=	99;
		END_IF
				
	99:	//Error
		
END_CASE

END_FUNCTION_BLOCK

// ---- POUs/Components/FB_FanBACnet.TcPOU
FUNCTION_BLOCK FB_FanBACnet
VAR_INPUT
	fSet	:	REAL;	//Setpoint 0-100%
END_VAR
VAR_OUTPUT
	bErr	:	BOOL;
END_VAR
VAR
	ManSetSpeed		:	FB_BACnet_RemoteAnalogOutput_EX;
	ManRelease		:	FB_BACnet_RemoteBinaryOutput_EX;
END_VAR

ManSetSpeed(RemoteDevice:=AHU_Bacnet.DevAHU,fPV:=fSet,bEnablePV:=TRUE);
ManRelease(RemoteDevice:=AHU_Bacnet.DevAHU,bPV:=TRUE,bEnablePV:=TRUE);
IF ManSetSpeed.bError OR ManRelease.bError	THEN
	bErr	:=	TRUE;
ELSE
	bErr	:=	FALSE;		
END_IF

END_FUNCTION_BLOCK

// ---- POUs/Components/FB_FanControl.TcPOU
FUNCTION_BLOCK FB_FanControl
VAR_INPUT
	fSpeed	:	REAL;		//Fan speed setpoint 0..100%
END_VAR
VAR
	fSpeedSetRaw  AT%Q*	: INT 	:=0; 	//Raw value for terminal => send to valve
END_VAR
VAR CONSTANT
		fFactor : REAL :=327.67;	// factor for calculating the terminal integer values (from percentage to int)
END_VAR

fSpeedSetRaw := REAL_TO_INT(fSpeed*fFactor);

END_FUNCTION_BLOCK

// ---- POUs/Components/FB_HydThrotCir.TcPOU
FUNCTION_BLOCK FB_HydThrotCir
VAR_INPUT
	//Pump
	iPump			:	I_Pump;
	//Valve
	iValve			:	I_Valve;
	//Temperatures
	iTempSup		:	I_TemperatureSensor;
	iTempRet		:	I_TemperatureSensor;
	//Controller
	iControl		:	I_HydraulicThrottlingControl;
END_VAR
VAR_OUTPUT
END_VAR
VAR
	eMode : E_ControlMode := E_ControlMode.Off;
END_VAR

PROPERTY Mode : E_ControlMode
GET
Mode := THIS^.eMode;
END_GET
SET
THIS^.eMode := Mode;
END_SET
END_PROPERTY

METHOD Run
VAR_INPUT
END_VAR
//Update temperatures
iTempSup.Run();
iTempRet.Run();

//Run components
iPump.Run();
iValve.Run();

//Run controller
iControl.Mode := eMode;
iControl.TemperatureSupAct := iTempRet.Temperature;
iControl.Run();

//Pump set properties
IF eMode = E_ControlMode.Off THEN
	iPump.SetOn := FALSE;
ELSE
	iPump.SetOn := TRUE;
END_IF
iPump.ControlMode := iControl.PumpMode;
iPump.Setpoint := iControl.PumpSet;

//Valve set properties
iValve.OpeningSetpoint := iControl.ValveSet;
END_METHOD

END_FUNCTION_BLOCK

// ---- POUs/Components/FB_JetNozzle1.TcPOU
FUNCTION_BLOCK FB_JetNozzle1
VAR_INPUT
END_VAR
VAR_OUTPUT
END_VAR
VAR
	//Properties
	bError 					: BOOL := FALSE;
	fAngleActual 			: REAL;
	fAngleSetpoint 			: REAL := 50;
	//Raw values
	nAngleActual AT %I*		: INT;
	nAngleSetpoint AT %Q* 	: INT;
END_VAR

PROPERTY AngleActual : REAL
GET
AngleActual := THIS^.fAngleActual;
END_GET
SET
THIS^.fAngleActual := AngleActual;
END_SET
END_PROPERTY

PROPERTY AngleSetpoint : REAL
GET
AngleSetpoint := THIS^.fAngleSetpoint;
END_GET
SET
THIS^.fAngleSetpoint := AngleSetpoint;
END_SET
END_PROPERTY

PROPERTY Error : BOOL
GET
Error := THIS^.bError;
END_GET
SET
THIS^.bError := Error;
END_SET
END_PROPERTY

METHOD Run
VAR_INPUT
END_VAR
//Read feedback for opening position
fAngleActual := FC_Current4_20Raw_TO_Percentage(nAngleActual);

//Write setpoint for opening position
nAngleSetpoint := FC_Percentage_TO_Current4_20Raw(fAngleSetpoint);
END_METHOD

END_FUNCTION_BLOCK

// ---- POUs/Components/FB_JetNozzle2.TcPOU
FUNCTION_BLOCK FB_JetNozzle2
VAR_INPUT
END_VAR
VAR_OUTPUT
END_VAR
VAR
	//Properties
	bError 					: BOOL := FALSE;
	fAngleActual 			: REAL;
	fAngleSetpoint 			: REAL := 50;
	//Raw values
	nAngleActual AT %I*		: INT;
	nAngleSetpoint AT %Q* 	: INT;
END_VAR

PROPERTY AngleActual : REAL
GET
AngleActual := THIS^.fAngleActual;
END_GET
SET
THIS^.fAngleActual := AngleActual;
END_SET
END_PROPERTY

PROPERTY AngleSetpoint : REAL
GET
AngleSetpoint := THIS^.fAngleSetpoint;
END_GET
SET
THIS^.fAngleSetpoint := AngleSetpoint;
END_SET
END_PROPERTY

PROPERTY Error : BOOL
GET
Error := THIS^.bError;
END_GET
SET
THIS^.bError := Error;
END_SET
END_PROPERTY

METHOD Run
VAR_INPUT
END_VAR
//Read feedback for opening position
fAngleActual := FC_Voltage2_10Raw_TO_Percentage(nAngleActual);

//Write setpoint for opening position
nAngleSetpoint := FC_Percentage_TO_Voltage2_10Raw(fAngleSetpoint);
END_METHOD

END_FUNCTION_BLOCK

// ---- POUs/Components/FC_Voltage2_10Raw_TO_Percentage.TcPOU
FUNCTION FC_Voltage2_10Raw_TO_Percentage : REAL
VAR_INPUT
	i : INT;
END_VAR
VAR
	f : REAL;
	nIntMax : INT := 32767;
	nIntMin : INT := 6553;
END_VAR

FC_Voltage2_10Raw_TO_Percentage := 100*INT_TO_REAL(i-nIntMin)/(nIntMax-nIntMin);

END_FUNCTION

// ---- POUs/Components/FC_Percentage_TO_Voltage2_10Raw.TcPOU
FUNCTION FC_Percentage_TO_Voltage2_10Raw : INT
VAR_INPUT
	f : REAL;
END_VAR
VAR
	nIntMax : INT := 32767;
	nIntMin : INT := 6553;
END_VAR

FC_Percentage_TO_Voltage2_10Raw := REAL_TO_INT(nIntMin + (f/100)*(nIntMax-nIntMin));

END_FUNCTION

// ---- POUs/Components/FB_PumpBACnet.TcPOU
FUNCTION_BLOCK FB_PumpBACnet
VAR_INPUT
	fSet		:	REAL	:=	100.0;	//Percentage of maximum
	Mode		:	E_PumpControlMode;
	//Control mode: 1 - CONST_SPEED, 5 - CONST_PRESSURE, 6 - CONST_DIFFPRESS, 7 - VAR_DIFFPRESS, 12 - TEMP_VARIABLE, 13 - CONST_CONTROL
END_VAR
VAR_OUTPUT
	stInfo			:	ST_PumpInfo;
	bInitSuccess	:	BOOL;
	bError			:	BOOL;
END_VAR
VAR
	fSetRaw		:	REAL;
	//BACnet client
	DevPump		:	FB_BACnet_RemoteDevice;
	//BACnet values
	Setpoint	:	FB_BACnet_RemoteAnalogOutput_EX;
	ContMode	:	FB_BACnet_RemoteMultiStateOutput_EX;
	PumpOn		:	FB_BACnet_RemoteBinaryOutput_EX;
	Operating	:	FB_BACnet_RemoteBinaryInput_EX;
	EstFlow		:	FB_BACnet_RemoteAnalogInput_EX;		//Estimated volume flow
	EstPressure	:	FB_BACnet_RemoteAnalogInput_EX;		//Estimated pressure difference
	Speed		:	FB_BACnet_RemoteAnalogInput_EX;
	Power_Act  	:	FB_BACnet_RemoteAnalogInput_EX;
	PumpError	:	FB_BACnet_RemoteBinaryInput_EX;
END_VAR

//Regular operation
PumpError(RemoteDevice:=DevPump,bPresentValue=>bError);	//Read pump error status
IF DevPump.bOperational THEN
	CASE  Mode OF
	
	E_PumpControlMode.NONE:
		PumpOn(RemoteDevice:=DevPump, bNullPV:= TRUE, bEnablePV:=TRUE);		//Release BACnet Value
		ContMode(RemoteDevice:=DevPump, bNullPV:= TRUE, bEnablePV:=TRUE);	//Release BACnet Value
	
  	E_PumpControlMode.OFF:
		PumpOn(RemoteDevice:=DevPump,bPV:=FALSE,bEnablePV:=TRUE);			// switch pump off
	
	ELSE
		PumpOn(RemoteDevice:=DevPump,bPV:=TRUE,bEnablePV:=TRUE);
		ContMode(RemoteDevice:=DevPump,nPV:=INT_TO_UDINT(Mode), bNullPV:= FALSE, bEnablePV:=TRUE);	//Set to appropriate control mode
	END_CASE
END_IF
//Error handling
IF (DevPump.bError) OR (Setpoint.bError) OR (PumpOn.bError) OR (bError) THEN
		PumpOn(RemoteDevice:=DevPump, bPV:=FALSE, bEnablePV:=TRUE);	//Deactivate Pump in Error
END_IF

//Write Setpoint value
Setpoint(RemoteDevice:=DevPump,fPV:=fSet,bEnablePV:=TRUE);	//Setpoint

//current values
EstFlow(RemoteDevice:=DevPump,fPresentValue=>stInfo.fVolFlow);
Speed(RemoteDevice:=DevPump,fPresentValue=>stInfo.fSpeed);
Power_Act(RemoteDevice:=DevPump,fPresentValue=>stInfo.fPower);
EstPressure(RemoteDevice:=DevPump,fPresentValue=>stInfo.fPressDiff);
Operating(RemoteDevice:=DevPump,bPresentValue=>stInfo.bOperating);

METHOD Init : BOOL
VAR_INPUT
END_VAR
//Init Device
DevPump(
	bReset:=FALSE,
	bAutoReset:=FALSE,
	bDisableWOC:=FALSE,
	bReSubscribeCOV:=FALSE,
	bAutoResubscribe:=FALSE,
	bTriggerWOC:=FALSE,
	bReload:=FALSE
);
IF DevPump.bOperational THEN
	ContMode(RemoteDevice:=DevPump,nPV:=INT_TO_UDINT(1),bEnablePV:=TRUE);	//Set to appropriate control mode
	//PumpOn(RemoteDevice:=DevPump,fPV:=1,bEnablePV:=TRUE);	//Activate Pump
	PumpOn(RemoteDevice:=DevPump,bPV:=TRUE,bEnablePV:=TRUE);	//Activate Pump
	IF (NOT ContMode.bError) AND (NOT PumpOn.bError) THEN
		bInitSuccess	:=	TRUE;
	END_IF
END_IF
bInitSuccess := TRUE;
END_METHOD

END_FUNCTION_BLOCK

// ---- POUs/Components/FB_PumpBACnet1.TcPOU
FUNCTION_BLOCK FB_PumpBACnet1 IMPLEMENTS I_Pump
VAR_INPUT CONSTANT
	fbClient : FB_BACnet_Client;
END_VAR
VAR_OUTPUT
END_VAR
VAR
	//Properties
	eControlMode : E_PumpControlMode := E_PumpControlMode.OFF;
	bError : BOOL;
	bOperating : BOOL;
	fPowerRating : REAL;
	fPressure : REAL;
	bSetOn : BOOL := FALSE;
	fSetpoint : REAL := 0;
	fSpeed : REAL;
	fVolumeFlow : REAL;	

	//BACnet parameters
	nPriority : BYTE := 12;
	
	//BACnet Mapping
	ContModeBAC		:	FB_BACnetRM_MO := (Client := fbClient, nObjectInstance :=0);		//Pump Control mode (speed, var/const pressure)
	ErrorBAC		:	FB_BACnetRM_BI := (Client := fbClient, nObjectInstance :=13);		//Error
	OperatingBAC	:	FB_BACnetRM_BI := (Client := fbClient, nObjectInstance :=0);		//Operation active/inactive
	PowerRatingBAC	:	FB_BACnetRM_AI := (Client := fbClient, nObjectInstance :=2);		//Current power
	PressureBAC		:	FB_BACnetRM_AI := (Client := fbClient, nObjectInstance :=1);		//Estimated pressure difference
	SetpointBAC		:	FB_BACnetRM_AO := (Client := fbClient, nObjectInstance :=0);		//Setpoint
	SetOnBAC		:	FB_BACnetRM_BO := (Client := fbClient, nObjectInstance :=0);		//Turn on/off
	SpeedBAC		:	FB_BACnetRM_AI := (Client := fbClient, nObjectInstance :=3);		//Estimated speed
	VolumeFlowBAC	:	FB_BACnetRM_AI := (Client := fbClient, nObjectInstance :=0);		//Estimated volume flow

END_VAR

PROPERTY ControlMode : E_PumpControlMode
GET
ControlMode := THIS^.eControlMode;
END_GET
SET
THIS^.eControlMode := ControlMode;
END_SET
END_PROPERTY

PROPERTY Error : BOOL
GET
Error := THIS^.bError;
END_GET
SET
THIS^.bError := Error;
END_SET
END_PROPERTY

PROPERTY Operating : BOOL
GET
Operating := THIS^.bOperating;
END_GET
SET
THIS^.bOperating := Operating;
END_SET
END_PROPERTY

PROPERTY PowerRating : REAL
GET
PowerRating := THIS^.fPowerRating;
END_GET
SET
THIS^.fPowerRating := PowerRating;
END_SET
END_PROPERTY

PROPERTY Pressure : REAL
GET
Pressure := THIS^.fPressure;
END_GET
SET
THIS^.fPressure := Pressure;
END_SET
END_PROPERTY

METHOD Run
//Run BACnet Client
fbClient();

//Read BACnet values
ErrorBAC(bPresentValue=>bError);
OperatingBAC(bPresentValue=>bOperating);
PowerRatingBAC(fPresentValue=>fPowerRating);
PressureBAC(fPresentValue=>fPressure);
SpeedBAC(fPresentValue=>fSpeed);
VolumeFlowBAC(fPresentValue=>fVolumeFlow);

//Write BACnet values
//Set pump values depending on defined ControlMode
IF eControlMode = E_PumpControlMode.OFF THEN
	//Set pump to off
	SetOnBAC(bPv:=FALSE,bEnablePv:=TRUE,nPriority:=nPriority);
	ContModeBAC(nPv:=eControlMode,bEnablePv:=TRUE,nPriority:=nPriority);
	SetpointBAC(fPv:=0,bEnablePv:=TRUE,nPriority:=nPriority);
ELSIF eControlMode = E_PumpControlMode.NONE THEN
	//Release
	SetOnBAC(bNullPv:=TRUE,nPriority:=nPriority); 	//Clear entry
	ContModeBAC(bNullPv:=TRUE,nPriority:=nPriority); //Clear entry
	SetpointBAC(bNullPv:=TRUE,nPriority:=nPriority); //Clear entry
ELSE
	//Set pump to on and set setpoint
	SetOnBAC(bPV:=TRUE,bEnablePv:=TRUE,nPriority:=nPriority);
	ContModeBAC(nPV:=eControlMode,bEnablePv:=TRUE,nPriority:=nPriority);
	SetpointBAC(fPV:=fSetpoint,bEnablePv:=TRUE,nPriority:=nPriority);
END_IF
END_METHOD

PROPERTY SetOn : BOOL
GET
SetOn := THIS^.bSetOn;
END_GET
SET
THIS^.bSetOn := SetOn;
END_SET
END_PROPERTY

PROPERTY Setpoint : REAL
GET
Setpoint := THIS^.fSetpoint;
END_GET
SET
THIS^.fSetpoint := Setpoint;
END_SET
END_PROPERTY

PROPERTY Speed : REAL
GET
Speed := THIS^.fSpeed;
END_GET
SET
THIS^.fSpeed := Speed;
END_SET
END_PROPERTY

PROPERTY VolumeFlow : REAL
GET
VolumeFlow := THIS^.fVolumeFlow;
END_GET
SET
THIS^.fVolumeFlow := VolumeFlow;
END_SET
END_PROPERTY

END_FUNCTION_BLOCK

// ---- POUs/Components/FB_PumpWiloIF.TcPOU
FUNCTION_BLOCK FB_PumpWiloIF
VAR_INPUT
	SetPoint 	AT %Q*	: REAL;  // Set point in %, depending on control mode; Connect with BacNet 'Bus Setpoint / Outputs / PresentValue'
END_VAR
VAR_OUTPUT
	mode		AT %I*	: UDINT;// Actual modes: n-c (const_speed) = 1, dp_c = 6, dp-v = 7; Connect with BacNet 'System Control Mode / Inputs / PresentValue'
	Speed 		AT %I*	: REAL;	// Actual Speed; Connect with 'Speed / Inputs / PresentValue'
	EstimFlow	AT %I*	: REAL;	// Estimated Flow; Connect with 'Estimated Flow / Inputs / PresentValue'
	dp			AT %I*	: REAL; // (Estimated) Pressure; Connect with '(Estimated) Pressure / Inputs / PresentValue'
	T			AT %I*	: REAL; // Medium Temperature; Connect with Bacnet 'Medium Temperature / Inputs /
	Operating	AT %I*	: WORD;	// Pump Operating; Connect with 'Status Pump is operating / Inputs / PresentValue'
	Power		AT %I*	: REAL;	//Power consumption; 'Power Rating / Inputs / PresentValue'
	Error		AT %I*	: WORD;	// Connect with 'Status Error Present / Inputs / PresentValue'
END_VAR
VAR	
	pumpOnSet	AT %Q*  : BOOL;  // True if pump is set on; Connect with BacNet 'Bus Command Pump on / Outputs / PresentValue'
	modeSet	 	AT %Q*	: UDINT; // modes: n-c (const_speed) = 1, dp_c = 6, dp-v = 7; Connect with BacNet 'Bus Control Mode / Outputs / PresentValue'

END_VAR

METHOD dp_c : BOOL
VAR_INPUT
END_VAR
modeSet := 6;
pumpOnSet := TRUE;
END_METHOD

METHOD dp_v : BOOL
VAR_INPUT
END_VAR
modeSet := 7;
pumpOnSet := TRUE;
END_METHOD

METHOD n_c : BOOL
VAR_INPUT
END_VAR
modeSet := 1;
pumpOnSet := TRUE;
END_METHOD

METHOD Off : BOOL
VAR_INPUT
END_VAR
pumpOnSet := False;
END_METHOD

END_FUNCTION_BLOCK

// ---- POUs/Components/FB_RoomControlUnit.TcPOU
FUNCTION_BLOCK FB_RoomControlUnit
VAR_INPUT
	fOffsetTemp :	REAL;
END_VAR
VAR_OUTPUT
	fPos		:	REAL;	//-100% - +100%
	bButton		:	BOOL;	//Button pressed?
	fTemp		:	REAL;	//Temperature
END_VAR
VAR
	nPosRaw		AT	%I*	:	INT;
	bButtonRaw	AT	%I*	:	BOOL;
	nTempRaw	AT	%I*	:	INT;
END_VAR
VAR CONSTANT
	fVal	:	REAL	:=	327.67;	//percentage to int
END_VAR

//TODO: Check which integer value corresponds to which position
bButton	:=	bButtonRaw;
fPos	:=	nPosRaw/fVal;
fTemp	:=	INT_TO_REAL(nTempRaw)/10 + fOffsetTemp;

END_FUNCTION_BLOCK

// ---- POUs/Components/FB_SenTempEL321x.TcPOU
FUNCTION_BLOCK FB_SenTempEL321x
VAR_INPUT
END_VAR
VAR_OUTPUT
	T : REAL;				// calculated temperature
END_VAR
VAR
	TempRaw  AT %I* : INT;  //Value from Terminal
		
END_VAR

T := INT_TO_REAL(TempRaw) / 10;

END_FUNCTION_BLOCK

// ---- POUs/Components/FB_TVJModbusMaster.TcPOU
FUNCTION_BLOCK FB_TVJModbusMaster
VAR_INPUT
END_VAR
VAR_OUTPUT
END_VAR
VAR
	fbModbusRTUMaster : ModbusRtuMaster_KL6x22B;	//Modbus RTU Master
	
	nUnitID			:	BYTE :=	0;	//Modbus device ID
	
	//Modbus Registers
	nRegSetpoint	:	WORD := 0;
	nRegForce		:	WORD := 1;
	nRegActual		:	WORD := 7;
	
	//Properties
	bError 			: 	BOOL := FALSE;
	fNominalVolFlow	: 	REAL := 8820;
	fVolFlowSet 	: 	REAL := 0;
	fVolFlowAct		: 	REAL;
	
	//Internal vars
	bFlagForce		:	BOOL := FALSE;
	bModErr 		: 	BOOL;
	ErrID 			: 	MODBUS_ERRORS;
	fRelFlowMax		:	WORD := 10000;
	fRelFlowMin		:	WORD := 2000;
	nForce			:	WORD := 0;
	fSetModbus		:	WORD := fRelFlowMin;
	sVolFlowAct		: 	WORD;
	
	//Timer
	Tim			:	TON;
	
	//State
	nState		:	INT	:= 1;
	
END_VAR

PROPERTY Error : Bool
GET
Error := THIS^.bError;
END_GET
SET
THIS^.bError := Error;
END_SET
END_PROPERTY

PROPERTY NominalVolumeFlow : REAL
GET
NominalVolumeFlow := THIS^.fNominalVolFlow;
END_GET
SET
THIS^.fNominalVolFlow := NominalVolumeFlow;
END_SET
END_PROPERTY

METHOD Run : BOOL
VAR_INPUT
END_VAR

VAR
	END_I: INT;
END_VAR
Tim(PT:=T#100MS,IN:=TRUE);
	IF Tim.Q THEN
		Tim(IN:=FALSE);

		CASE nState OF
			//Force or release force
			1: //Initialize writing force or release
				IF NOT fbModbusRTUMaster.BUSY THEN
					//IF setpoint is 0, force close ELSE release force mode
					IF fVolFlowSet = 0 OR bFlagForce = TRUE THEN
						//Force close
						nForce := 2;
						//Initialize writing process
						fbModbusRTUMaster.WriteSingleRegister(	UnitID		:=	nUnitID,				//Modbus ID of device
																MBAddr		:=	nRegForce,				//Register address,
																Quantity	:=	1,						//Number of registers to be written
																pMemoryAddr	:=	ADR(nForce),			//Pointer to write data
																cbLength	:=	SIZEOF(fVolFlowSet),	//Size of write data
																Timeout		:=	T#5S,					//Time to wait for the slave to respond
																Execute		:=	TRUE
															);
					ELSE
						//Release force close
						nForce := 0;
						//Initialize writing process
						fbModbusRTUMaster.WriteSingleRegister(	UnitID		:=	nUnitID,				//Modbus ID of device
																MBAddr		:=	nRegForce,				//Register address,
																Quantity	:=	1,						//Number of registers to be written
																pMemoryAddr	:=	ADR(nForce),			//Pointer to write data
																cbLength	:=	SIZEOF(fVolFlowSet),	//Size of write data
																Timeout		:=	T#5S,					//Time to wait for the slave to respond
																Execute		:=	TRUE
															);
					END_IF
				END_IF
				nState := 2;
				Run := FALSE;
				
			2:	//Finish writing force or release
				fbModbusRTUMaster.WriteSingleRegister(Execute:=FALSE, Error=>bModErr, ErrorID=>ErrID);
				IF NOT fbModbusRTUMaster.BUSY THEN
					nState := 3;
				END_IF
				Run := FALSE;
				
			3:	//Setpoint writing
				IF NOT fbModbusRTUMaster.BUSY THEN
					//Check operational limits
					IF fVolFlowSet < fRelFlowMin/fRelFlowMax*fNominalVolFlow THEN
						fVolFlowSet := fRelFlowMin/fRelFlowMax*fNominalVolFlow; //Set to minimum allowed volume flow
					ELSIF fVolFlowSet > fNominalVolFlow THEN
						fVolFlowSet := fNominalVolFlow; //Set to maximum allowed volumen flow
					ELSE
						//do nothing
					END_IF
					//Write setpoint
					//fSetModbus := REAL_TO_WORD(fRelFlowMax*(fVolFlowSet-(fRelFlowMin/fRelFlowMax*fNominalVolFlow))/(fNominalVolFlow-fRelFlowMin));
					fSetModbus := REAL_TO_WORD(fRelFlowMax*fVolFlowSet/fNominalVolFlow);
					//Initialize writing process
					fbModbusRTUMaster.WriteSingleRegister(	UnitID		:=	nUnitID,				//Modbus ID of device
															MBAddr		:=	nRegSetpoint,			//Register address
															Quantity	:=	1,						//Number of registers to be written
															pMemoryAddr	:=	ADR(fSetModbus),		//Pointer to write data
															cbLength	:=	SIZEOF(fSetModbus),		//Size of write data
															Timeout		:=	T#5S,					//Time to wait for the slave to respond
															Execute		:=	TRUE
														);
				END_IF
				nState := 4;
				Run := FALSE;

			4: //Finish writing	
				fbModbusRTUMaster.WriteSingleRegister(Execute:=FALSE, Error=>bModErr, ErrorID=>ErrID);
				IF NOT fbModbusRTUMaster.BUSY THEN
					nState := 5;
				END_IF
				Run := FALSE;
					
			5: //Start reading
				IF NOT fbModbusRTUMaster.BUSY THEN
					//Initialize reading process
					fbModbusRTUMaster.ReadRegs(	UnitID		:=	nUnitID,				//Modbus ID of device
												MBAddr		:=	nRegActual,				//Register address
												Quantity	:=	1,						//Number of registers to be read
												pMemoryAddr	:=	ADR(sVolFlowAct),		//Pointer to read data
												cbLength	:=	SIZEOF(sVolFlowAct),	//Size of read data
												Timeout		:=	T#5S,					//Time to wait for the slave to respond
												Execute		:=	TRUE
												);
				ELSE
					//do nothing
				END_IF
				nState := 6;
				Run := FALSE;
				
			6: //Finish reading
				fbModbusRTUMaster.ReadRegs(Execute:=FALSE, Error=>bModErr, ErrorID=>ErrID);
				IF NOT fbModbusRTUMaster.BUSY THEN
					fVolFlowAct := WORD_TO_REAL(sVolFlowAct);
					nState := 1;
					Run := TRUE;
				ELSE
					Run := FALSE;
				END_IF
				
		END_CASE
		
END_IF
END_METHOD

PROPERTY UnitID : BYTE
GET
UnitID := THIS^.nUnitID;
END_GET
SET
THIS^.nUnitID := UnitID;
END_SET
END_PROPERTY

PROPERTY VolumeFlowActual : REAL
GET
VolumeFlowActual := THIS^.fVolFlowAct;
END_GET
SET
THIS^.fVolFlowAct := VolumeFlowActual;
END_SET
END_PROPERTY

PROPERTY VolumeFlowSetpoint : REAL
GET
VolumeFlowSetpoint := THIS^.fVolFlowSet;
END_GET
SET
THIS^.fVolFlowSet := VolumeFlowSetpoint;
END_SET
END_PROPERTY

END_FUNCTION_BLOCK

// ---- POUs/Components/FB_TVRModbusMaster.TcPOU
FUNCTION_BLOCK FB_TVRModbusMaster
VAR_INPUT
END_VAR
VAR_OUTPUT
END_VAR
VAR
	fbModbusRTUMaster : ModbusRtuMaster_KL6x22B;	//Modbus RTU Master
	
	nUnitID			:	BYTE :=	0;	//Modbus device ID
	
	//Modbus Registers
	nRegSetpoint	:	WORD := 0;
	nRegForce		:	WORD := 1;
	nRegActual		:	WORD := 7;
	
	//Properties
	bError 			: 	BOOL := FALSE;
	fNominalVolFlow	: 	REAL := 3690;
	fVolFlowSet 	: 	REAL := 0;
	fVolFlowAct		: 	REAL;
	
	//Internal vars
	bFlagForce		:	BOOL := FALSE;
	bModErr 		: 	BOOL;
	ErrID 			: 	MODBUS_ERRORS;
	fRelFlowMax		:	WORD := 10000;
	fRelFlowMin		:	WORD := 1024;
	nForce			:	WORD := 0;
	fSetModbus		:	WORD := fRelFlowMin;
	sVolFlowAct		: 	WORD;
	
	//Timer
	Tim			:	TON;
	
	//State
	nState		:	INT	:= 1;
	
END_VAR

PROPERTY Error : Bool
GET
Error := THIS^.bError;
END_GET
SET
THIS^.bError := Error;
END_SET
END_PROPERTY

PROPERTY NominalVolumeFlow : REAL
GET
NominalVolumeFlow := THIS^.fNominalVolFlow;
END_GET
SET
THIS^.fNominalVolFlow := NominalVolumeFlow;
END_SET
END_PROPERTY

METHOD Run : BOOL
VAR_INPUT
END_VAR

VAR
	END_I: INT;
END_VAR
Tim(PT:=T#100MS,IN:=TRUE);
	IF Tim.Q THEN
		Tim(IN:=FALSE);

		CASE nState OF
			//Force or release force
			1: //Initialize writing force or release
				IF NOT fbModbusRTUMaster.BUSY THEN
					//IF setpoint is 0, force close ELSE release force mode
					IF fVolFlowSet = 0 OR bFlagForce = TRUE THEN
						//Force close
						nForce := 2;
						//Initialize writing process
						fbModbusRTUMaster.WriteSingleRegister(	UnitID		:=	nUnitID,				//Modbus ID of device
																MBAddr		:=	nRegForce,				//Register address,
																Quantity	:=	1,						//Number of registers to be written
																pMemoryAddr	:=	ADR(nForce),			//Pointer to write data
																cbLength	:=	SIZEOF(fVolFlowSet),	//Size of write data
																Timeout		:=	T#5S,					//Time to wait for the slave to respond
																Execute		:=	TRUE
															);
					ELSE
						//Release force close
						nForce := 0;
						//Initialize writing process
						fbModbusRTUMaster.WriteSingleRegister(	UnitID		:=	nUnitID,				//Modbus ID of device
																MBAddr		:=	nRegForce,				//Register address,
																Quantity	:=	1,						//Number of registers to be written
																pMemoryAddr	:=	ADR(nForce),			//Pointer to write data
																cbLength	:=	SIZEOF(fVolFlowSet),	//Size of write data
																Timeout		:=	T#5S,					//Time to wait for the slave to respond
																Execute		:=	TRUE
															);
					END_IF
				END_IF
				nState := 2;
				Run := FALSE;
				
			2:	//Finish writing force or release
				fbModbusRTUMaster.WriteSingleRegister(Execute:=FALSE, Error=>bModErr, ErrorID=>ErrID);
				IF NOT fbModbusRTUMaster.BUSY THEN
					nState := 3;
				END_IF
				Run := FALSE;
				
			3:	//Setpoint writing
				IF NOT fbModbusRTUMaster.BUSY THEN
					//Check operational limits
					IF fVolFlowSet < fRelFlowMin/fRelFlowMax*fNominalVolFlow THEN
						fVolFlowSet := fRelFlowMin/fRelFlowMax*fNominalVolFlow; //Set to minimum allowed volume flow
					ELSIF fVolFlowSet > fNominalVolFlow THEN
						fVolFlowSet := fNominalVolFlow; //Set to maximum allowed volumen flow
					ELSE
						//do nothing
					END_IF
					//Write setpoint
					//fSetModbus := REAL_TO_WORD(fRelFlowMax*(fVolFlowSet-(fRelFlowMin/fRelFlowMax*fNominalVolFlow))/(fNominalVolFlow-fRelFlowMin));
					fSetModbus := REAL_TO_WORD(fRelFlowMax*fVolFlowSet/fNominalVolFlow);
					//Initialize writing process
					fbModbusRTUMaster.WriteSingleRegister(	UnitID		:=	nUnitID,				//Modbus ID of device
															MBAddr		:=	nRegSetpoint,			//Register address
															Quantity	:=	1,						//Number of registers to be written
															pMemoryAddr	:=	ADR(fSetModbus),		//Pointer to write data
															cbLength	:=	SIZEOF(fSetModbus),		//Size of write data
															Timeout		:=	T#5S,					//Time to wait for the slave to respond
															Execute		:=	TRUE
														);
				END_IF
				nState := 4;
				Run := FALSE;

			4: //Finish writing	
				fbModbusRTUMaster.WriteSingleRegister(Execute:=FALSE, Error=>bModErr, ErrorID=>ErrID);
				IF NOT fbModbusRTUMaster.BUSY THEN
					nState := 5;
				END_IF
				Run := FALSE;
					
			5: //Start reading
				IF NOT fbModbusRTUMaster.BUSY THEN
					//Initialize reading process
					fbModbusRTUMaster.ReadRegs(	UnitID		:=	nUnitID,				//Modbus ID of device
												MBAddr		:=	nRegActual,				//Register address
												Quantity	:=	1,						//Number of registers to be read
												pMemoryAddr	:=	ADR(sVolFlowAct),		//Pointer to read data
												cbLength	:=	SIZEOF(sVolFlowAct),	//Size of read data
												Timeout		:=	T#5S,					//Time to wait for the slave to respond
												Execute		:=	TRUE
												);
				ELSE
					//do nothing
				END_IF
				nState := 6;
				Run := FALSE;
				
			6: //Finish reading
				fbModbusRTUMaster.ReadRegs(Execute:=FALSE, Error=>bModErr, ErrorID=>ErrID);
				IF NOT fbModbusRTUMaster.BUSY THEN
					fVolFlowAct := WORD_TO_REAL(sVolFlowAct);
					nState := 1;
					Run := TRUE;
				ELSE
					Run := FALSE;
				END_IF
				
		END_CASE
		
END_IF
END_METHOD

PROPERTY UnitID : BYTE
GET
UnitID := THIS^.nUnitID;
END_GET
SET
THIS^.nUnitID := UnitID;
END_SET
END_PROPERTY

PROPERTY VolumeFlowActual : REAL
GET
VolumeFlowActual := THIS^.fVolFlowAct;
END_GET
SET
THIS^.fVolFlowAct := VolumeFlowActual;
END_SET
END_PROPERTY

PROPERTY VolumeFlowSetpoint : REAL
GET
VolumeFlowSetpoint := THIS^.fVolFlowSet;
END_GET
SET
THIS^.fVolFlowSet := VolumeFlowSetpoint;
END_SET
END_PROPERTY

END_FUNCTION_BLOCK

// ---- POUs/Components/FB_ValveBACnet.TcPOU
FUNCTION_BLOCK FB_ValveBACnet IMPLEMENTS I_Valve
VAR_INPUT
	//fbClient : FB_BACnet_Client;
END_VAR
VAR_OUTPUT
END_VAR
VAR
	//Properties
	bError 					: BOOL := FALSE;
	fOpeningActual 			: REAL;
	fOpeningSetpoint 		: REAL := 0;

(*	
	//BACnet parameters
	nPriority : BYTE := 12;
	
	//BACnet Mapping
	//Only one Client of the same DeviceInstance
*)
END_VAR

PROPERTY Error : BOOL
GET
Error := THIS^.bError;
END_GET
SET
THIS^.bError := Error;
END_SET
END_PROPERTY

PROPERTY OpeningActual : REAL
GET
OpeningActual := THIS^.fOpeningActual;
END_GET
SET
THIS^.fOpeningActual := OpeningActual;
END_SET
END_PROPERTY

PROPERTY OpeningSetpoint : REAL
GET
OpeningSetpoint := THIS^.fOpeningSetpoint;
END_GET
SET
THIS^.fOpeningSetpoint := OpeningSetpoint;
END_SET
END_PROPERTY

METHOD Run
(*
//Run BACnet client
fbClient();

//Read BACnet values
ReheaterValActBAC(fPresentValue=>fOpeningActual);

//Write BACnet values
ReheaterValSetBAC(fPV:=fOpeningSetpoint,bEnablePv:=TRUE,nPriority:=nPriority);
*)
END_METHOD

END_FUNCTION_BLOCK

// ---- POUs/Components/FB_Valve_0_10V.TcPOU
FUNCTION_BLOCK FB_Valve_0_10V IMPLEMENTS I_Valve
VAR_INPUT
END_VAR
VAR_OUTPUT
END_VAR
VAR
		//Properties
	bError : BOOL := FALSE;
	fOpeningActual : REAL;
	fOpeningSetpoint : REAL := 0;
	//Raw values
	nOpeningSet AT %Q* : INT;
	nOpeningAct AT %I* : INT;
END_VAR

{warning 'Eigenschaftenimplementierung hinzufügen'}
PROPERTY Error : BOOL
GET
Error := THIS^.bError;
END_GET
SET
THIS^.bError := Error;
END_SET
END_PROPERTY

{warning 'Eigenschaftenimplementierung hinzufügen'}
PROPERTY OpeningActual : REAL
GET
OpeningActual := THIS^.fOpeningActual;
END_GET
SET
THIS^.fOpeningActual := OpeningActual;
END_SET
END_PROPERTY

{warning 'Eigenschaftenimplementierung hinzufügen'}
PROPERTY OpeningSetpoint : REAL
GET
OpeningSetpoint := THIS^.fOpeningSetpoint;
END_GET
SET
THIS^.fOpeningSetpoint := OpeningSetpoint;
END_SET
END_PROPERTY

{warning 'Methodenimplementierung hinzufügen'}
METHOD Run
//Read feedback for opening position
fOpeningActual := FC_Voltage0_10Raw_TO_Percentage(nOpeningAct);

//Write setpoint for opening position
nOpeningSet := FC_Percentage_TO_Voltage0_10Raw(fOpeningSetpoint);
END_METHOD

END_FUNCTION_BLOCK

// ---- POUs/Components/FC_Voltage0_10Raw_TO_Percentage.TcPOU
FUNCTION FC_Voltage0_10Raw_TO_Percentage : REAL
VAR_INPUT
	i : INT;
END_VAR
VAR
	f : REAL;
	nIntMax : INT := 32767;
	nIntMin : INT := 0;
END_VAR

FC_Voltage0_10Raw_TO_Percentage := 100*INT_TO_REAL(i-nIntMin)/(nIntMax-nIntMin);

END_FUNCTION

// ---- POUs/Components/FC_Percentage_TO_Voltage0_10Raw.TcPOU
FUNCTION FC_Percentage_TO_Voltage0_10Raw : INT
VAR_INPUT
	f : REAL;
END_VAR
VAR
	nIntMax : INT := 32767;
	nIntMin : INT := 0;
END_VAR

FC_Percentage_TO_Voltage0_10Raw := REAL_TO_INT(nIntMin + (f/100)*(nIntMax-nIntMin));

END_FUNCTION

// ---- POUs/Components/FB_Valve_2_10V.TcPOU
FUNCTION_BLOCK FB_Valve_2_10V IMPLEMENTS I_Valve
VAR_INPUT
END_VAR
VAR_OUTPUT
END_VAR
VAR
	//Properties
	bError : BOOL := FALSE;
	fOpeningActual : REAL;
	fOpeningSetpoint : REAL := 0;
	//Raw values
	nOpeningSet AT %Q* : INT;
	nOpeningAct AT %I* : INT;
END_VAR

PROPERTY Error : BOOL
GET
Error := THIS^.bError;
END_GET
SET
THIS^.bError := Error;
END_SET
END_PROPERTY

PROPERTY OpeningActual : REAL
GET
OpeningActual := THIS^.fOpeningActual;
END_GET
SET
THIS^.fOpeningActual := OpeningActual;
END_SET
END_PROPERTY

PROPERTY OpeningSetpoint : REAL
GET
OpeningSetpoint := THIS^.fOpeningSetpoint;
END_GET
SET
THIS^.fOpeningSetpoint := OpeningSetpoint;
END_SET
END_PROPERTY

METHOD Run
//Read feedback for opening position
fOpeningActual := FC_Voltage2_10Raw_TO_Percentage(nOpeningAct);

//Write setpoint for opening position
nOpeningSet := FC_Percentage_TO_Voltage2_10Raw(fOpeningSetpoint);
END_METHOD

END_FUNCTION_BLOCK

// ---- POUs/Components/FB_VFCModbus1.TcPOU
FUNCTION_BLOCK FB_VFCModbus1 IMPLEMENTS I_VolumeFlowController
VAR_INPUT CONSTANT
	fbModbusMaster	:	POINTER TO FB_TVRModbusMaster;
	nUnitID			:	BYTE;
END_VAR
VAR_OUTPUT
END_VAR
VAR
	//Properties
	bError 			: 	BOOL := FALSE;
	fNominalVolFlow	: 	REAL := 3690;
	fVolFlowSet 	: 	REAL := 0;
	fVolFlowAct		: 	REAL;
	
	bFinish 		:	BOOL;
	
END_VAR

PROPERTY Error : BOOL
GET
Error := THIS^.bError;
END_GET
SET
THIS^.bError := Error;
END_SET
END_PROPERTY

PROPERTY NominalVolumeFlow : REAL
GET
NominalVolumeFlow := THIS^.fNominalVolFlow;
END_GET
SET
THIS^.fNominalVolFlow := NominalVolumeFlow;
END_SET
END_PROPERTY

METHOD Run : BOOL
//Write properties to master
fbModbusMaster^.NominalVolumeFlow := fNominalVolFlow;
fbModbusMaster^.VolumeFlowSetpoint := fVolFlowSet;
fbModbusMaster^.UnitID := nUnitID;

//Execute modbus master
bFinish := fbModbusMaster^.Run();

//Read properties from master
bError := fbModbusMaster^.Error;
IF bFinish THEN
	fVolFlowAct := fbModbusMaster^.VolumeFlowActual;
END_IF

Run := bFinish;
END_METHOD

PROPERTY UnitID : BYTE
GET
UnitID := THIS^.nUnitID;
END_GET
SET
THIS^.nUnitID := UnitID;
END_SET
END_PROPERTY

PROPERTY VolumeFlowActual : REAL
GET
VolumeFlowActual := THIS^.fVolFlowAct;
END_GET
SET
THIS^.fVolFlowAct := VolumeFlowActual;
END_SET
END_PROPERTY

PROPERTY VolumeFlowSetpoint : REAL
GET
VolumeFlowSetpoint := THIS^.fVolFlowSet;
END_GET
SET
THIS^.fVolFlowSet := VolumeFlowSetpoint;
END_SET
END_PROPERTY

END_FUNCTION_BLOCK

// ---- POUs/Components/FB_VFCModbus2.TcPOU
FUNCTION_BLOCK FB_VFCModbus2 IMPLEMENTS I_VolumeFlowController
VAR_INPUT CONSTANT
	fbModbusMaster	:	POINTER TO FB_TVJModbusMaster;
	nUnitID			:	BYTE;
END_VAR
VAR_OUTPUT
END_VAR
VAR
	//Properties
	bError 			: 	BOOL := FALSE;
	fNominalVolFlow	: 	REAL := 8820;
	fVolFlowSet 	: 	REAL := 0;
	fVolFlowAct		: 	REAL;
	
	bFinish 		:	BOOL;
	
END_VAR

PROPERTY Error : BOOL
GET
Error := THIS^.bError;
END_GET
SET
THIS^.bError := Error;
END_SET
END_PROPERTY

PROPERTY NominalVolumeFlow : REAL
GET
NominalVolumeFlow := THIS^.fNominalVolFlow;
END_GET
SET
THIS^.fNominalVolFlow := NominalVolumeFlow;
END_SET
END_PROPERTY

METHOD Run : BOOL
//Write properties to master
fbModbusMaster^.NominalVolumeFlow := fNominalVolFlow;
fbModbusMaster^.VolumeFlowSetpoint := fVolFlowSet;
fbModbusMaster^.UnitID := nUnitID;

//Execute modbus master
bFinish := fbModbusMaster^.Run();

//Read properties from master
bError := fbModbusMaster^.Error;
IF bFinish THEN
	fVolFlowAct := fbModbusMaster^.VolumeFlowActual;
END_IF

Run := bFinish;
END_METHOD

PROPERTY UnitID : BYTE
GET
UnitID := THIS^.nUnitID;
END_GET
SET
THIS^.nUnitID := UnitID;
END_SET
END_PROPERTY

PROPERTY VolumeFlowActual : REAL
GET
VolumeFlowActual := THIS^.fVolFlowAct;
END_GET
SET
THIS^.fVolFlowAct := VolumeFlowActual;
END_SET
END_PROPERTY

PROPERTY VolumeFlowSetpoint : REAL
GET
VolumeFlowSetpoint := THIS^.fVolFlowSet;
END_GET
SET
THIS^.fVolFlowSet := VolumeFlowSetpoint;
END_SET
END_PROPERTY

END_FUNCTION_BLOCK

// ---- POUs/Components/FB_VVS_JN.TcPOU
FUNCTION_BLOCK FB_VVS_JN
VAR_INPUT
	fSet	:	ARRAY [1..10] OF REAL;	//Volume flow setpoint for each nozzle
	Init	:	BOOL;
END_VAR
VAR_OUTPUT
	fAct	:	ARRAY [1..10] OF ST_JNData;	//Actual volume flows
	InitSuccess	:	BOOL;
END_VAR
VAR	
	Step	:	INT		:=	1;
	i		:	USINT	:=	1;
	
	i_init	:	USINT	:=	1;
	Step_init	:	INT	:=	1;
	
	//Volume flow in percentage
	fVolFlowNorm	:	REAL	:=	3690;
	fVolFlowMin		:	REAL;
	fPercMax		:	WORD		:=	10000;
	fPercMin		:	WORD		:=	1024;
	fSetPerc		:	ARRAY[1..10] OF WORD;
	indVolFlow		:	INT;
	sErrMess		:	STRING;
	
	nZwang	:	WORD	:=	2;
	bZwang	:	Array[1..10] of  BOOL;
	
	//Modbus masters
	fbModK7		:	ModbusRtuMaster_KL6x22B;	//Nozzles 1,3,5,7 on terminal 7
	fbModK8		:	ModbusRtuMaster_KL6x22B;	//Nozzles 2,4,6,8,9,10 on terminal 8
	bModErr		:	BOOL;
	ErrID		:	MODBUS_ERRORS;
	
END_VAR

IF Init THEN	//Remove control override
	CASE Step_init OF
	
	1:
	nZwang	:=	0;
	IF (i_init=1) OR (i_init=3) OR (i_init=5) OR (i_init=7) THEN
		fbModK7.WriteSingleRegister(
			UnitID		:=	i_init,	//Modbus address of slave
			MBAddr		:=	1,	//Register address
			Quantity	:=	1,	//Number of registers to be written
			pMemoryAddr	:=	ADR(nZwang),		//Pointer to write data
			cbLength	:=	SIZEOF(nZwang),	//Size of write data
			Timeout		:=	T#5S,				//Time to wait for the slave to respond
			Execute		:=	TRUE
		);
	ELSE
		fbModK8.WriteSingleRegister(
			UnitID		:=	i_init,	//Modbus address of slave
			MBAddr		:=	1,	//Register address
			Quantity	:=	1,	//Number of registers to be written
			pMemoryAddr	:=	ADR(nZwang),		//Pointer to write data
			cbLength	:=	SIZEOF(nZwang),	//Size of write data
			Timeout		:=	T#5S,				//Time to wait for the slave to respond
			Execute		:=	TRUE
		);
	END_IF
	Step_init	:=	2;
	
	2:
	IF (i_init=1) OR (i_init=3) OR (i_init=5) OR (i_init=7) THEN
		fbModK7.WriteSingleRegister(Execute:=FALSE, Error=>bModErr, ErrorID=>ErrID);
		IF NOT fbModK7.BUSY THEN
			bZwang[i_init]	:=	FALSE;
			i_init		:=	i_init	+ 1;
			Step_init	:=	1;
			IF i_init > 10 THEN
				i_init	:=	1;
				Step_init :=	1;
				Init	:=	FALSE;
				InitSuccess	:=	TRUE;
			END_IF
		END_IF
	ELSE
		fbModK8.WriteSingleRegister(Execute:=FALSE, Error=>bModErr, ErrorID=>ErrID);
		IF NOT fbModK8.BUSY THEN
			bZwang[i_init]	:=	FALSE;
			i_init		:=	i_init	+ 1;
			Step_init	:=	1;
			IF i_init > 10 THEN
				i_init	:=	1;
				Step_init :=	1;
				Init	:=	FALSE;
				InitSuccess	:=	TRUE;
			END_IF
		END_IF
	END_IF

	END_CASE
ELSE

	fVolFlowMin	:=	fVolFlowNorm*fPercMin/10000;
	FOR indVolFlow := 1 TO 10 DO
		fAct[indVolFlow].SetFlow	:=	fSet[indVolFlow];
		fSetPerc[indVolFlow]	:=	REAL_TO_WORD(10000*(fSet[indVolFlow]-fVolFlowMin)/(fVolFlowNorm-fVolFlowMin)); //in hundreds of a percent between min and max
		IF fSet[indVolFlow] = 0 THEN
			sErrMess	:=	'Force Close';
			fSetPerc[indVolFlow]	:=	65535;	//Zwangssteuerung aus
		ELSIF fSetPerc[indVolFlow] > fPercMax THEN
			sErrMess	:=	'Requested volume flow larger than maximum. Setting value to maximum.';
			fSetPerc[indVolFlow]	:=	fPercMax;
		ELSIF fSetPerc[indVolFlow] < 0 AND fSet[indVolFlow] <> 0 THEN
			sErrMess	:=	'Requested volume flow smaller than minimum. Setting value to minimum.';
			fSetPerc[indVolFlow]	:=	0;		
		ELSE
			sErrMess	:=	'';
		END_IF
		fAct[indVolFlow].SetPerc	:=	fSetPerc[indVolFlow];
	END_FOR
	
	
	CASE Step OF
		
		1:	//start writing setpoint to nozzle
			IF fSetPerc[i] = 65535 THEN
				Step	:=	20;	//Control override
				bZwang[i]	:=	TRUE;
			ELSE
				IF bZwang[i] THEN
					Step :=	30;
				ELSE
					IF (i=1) OR (i=3) OR (i=5) OR (i=7) THEN
						fbModK7.WriteSingleRegister(
							UnitID		:=	i,	//Modbus address of slave
							MBAddr		:=	0,	//Register address
							Quantity	:=	1,	//Number of registers to be written
							pMemoryAddr	:=	ADR(fSetPerc[i]),		//Pointer to write data
							cbLength	:=	SIZEOF(fSetPerc[i]),	//Size of write data
							Timeout		:=	T#5S,				//Time to wait for the slave to respond
							Execute		:=	TRUE
						);
					ELSE
						fbModK8.WriteSingleRegister(
							UnitID		:=	i,	//Modbus address of slave
							MBAddr		:=	0,	//Register address
							Quantity	:=	1,	//Number of registers to be written
							pMemoryAddr	:=	ADR(fSetPerc[i]),		//Pointer to write data
							cbLength	:=	SIZEOF(fSetPerc[i]),	//Size of write data
							Timeout		:=	T#5S,				//Time to wait for the slave to respond
							Execute		:=	TRUE
						);
					END_IF
				Step	:=	2;
				END_IF
			END_IF
			
		2:	//finish writing process
			IF (i=1) OR (i=3) OR (i=5) OR (i=7) THEN
				fbModK7.WriteSingleRegister(Execute:=FALSE, Error=>bModErr, ErrorID=>ErrID);
				IF NOT fbModK7.BUSY THEN
					Step	:=	3;	//go to next step when writing process has finished
				END_IF
				IF fbModK7.Error THEN
					Step	:=	99;
				END_IF
			ELSE
				fbModK8.WriteSingleRegister(Execute:=FALSE, Error=>bModErr, ErrorID=>ErrID);
				IF NOT fbModK8.BUSY THEN
					Step	:=	3;	//go to next step when writing process has finished
				END_IF
				IF fbModK8.Error THEN
					Step	:=	99;
				END_IF
			END_IF
			
		3:	//start reading relative position
			IF (i=1) OR (i=3) OR (i=5) OR (i=7) THEN
				fbModK7.ReadRegs(
					UnitID		:=	i,	//Modbus address of slave
					MBAddr		:=	4,	//Register address
					Quantity	:=	1,	//Number of registers to be read
					pMemoryAddr	:=	ADR(fAct[i].PosRel),		//Pointer to read data
					cbLength	:=	SIZEOF(fAct[i].PosRel),	//Size of read data
					Timeout		:=	T#5S,				//Time to wait for the slave to respond
					Execute		:=	TRUE
				);
			ELSE
				fbModK8.ReadRegs(
					UnitID		:=	i,	//Modbus address of slave
					MBAddr		:=	4,	//Register address
					Quantity	:=	1,	//Number of registers to be read
					pMemoryAddr	:=	ADR(fAct[i].PosRel),		//Pointer to read data
					cbLength	:=	SIZEOF(fAct[i].PosRel),	//Size of read data
					Timeout		:=	T#5S,				//Time to wait for the slave to respond
					Execute		:=	TRUE
				);
			END_IF
			Step	:=	4;
			
		4:	//finish reading process
			IF (i=1) OR (i=3) OR (i=5) OR (i=7) THEN
				fbModK7.ReadRegs(Execute:=FALSE, Error=>bModErr, ErrorID=>ErrID);
				IF NOT fbModK7.BUSY THEN
					Step	:=	5;	//go to next step when reading process has finished
				END_IF
				IF fbModK7.Error THEN
					Step	:=	99;
				END_IF
			ELSE
				fbModK8.ReadRegs(Execute:=FALSE, Error=>bModErr, ErrorID=>ErrID);
				IF NOT fbModK8.BUSY THEN
					Step	:=	5;	//go to next step when reading process has finished
				END_IF
				IF fbModK8.Error THEN
					Step	:=	99;
				END_IF
			END_IF
			
		5:	//start reading absolute position
			IF (i=1) OR (i=3) OR (i=5) OR (i=7) THEN
				fbModK7.ReadRegs(
					UnitID		:=	i,	//Modbus address of slave
					MBAddr		:=	5,	//Register address
					Quantity	:=	1,	//Number of registers to be read
					pMemoryAddr	:=	ADR(fAct[i].PosAbs),		//Pointer to read data
					cbLength	:=	SIZEOF(fAct[i].PosAbs),	//Size of read data
					Timeout		:=	T#5S,				//Time to wait for the slave to respond
					Execute		:=	TRUE
				);
			ELSE
				fbModK8.ReadRegs(
					UnitID		:=	i,	//Modbus address of slave
					MBAddr		:=	5,	//Register address
					Quantity	:=	1,	//Number of registers to be read
					pMemoryAddr	:=	ADR(fAct[i].PosAbs),		//Pointer to read data
					cbLength	:=	SIZEOF(fAct[i].PosAbs),	//Size of read data
					Timeout		:=	T#5S,				//Time to wait for the slave to respond
					Execute		:=	TRUE
				);
			END_IF
			Step	:=	6;
			
		6:	//finish reading process
			IF (i=1) OR (i=3) OR (i=5) OR (i=7) THEN
				fbModK7.ReadRegs(Execute:=FALSE, Error=>bModErr, ErrorID=>ErrID);
				IF NOT fbModK7.BUSY THEN
					Step	:=	7;	//go to next step when reading process has finished
				END_IF
				IF fbModK7.Error THEN
					Step	:=	99;
				END_IF
			ELSE
				fbModK8.ReadRegs(Execute:=FALSE, Error=>bModErr, ErrorID=>ErrID);
				IF NOT fbModK8.BUSY THEN
					Step	:=	7;	//go to next step when reading process has finished
				END_IF
				IF fbModK8.Error THEN
					Step	:=	99;
				END_IF
			END_IF
		
		7:	//start reading relative volume flow
			IF (i=1) OR (i=3) OR (i=5) OR (i=7) THEN
				fbModK7.ReadRegs(
					UnitID		:=	i,	//Modbus address of slave
					MBAddr		:=	6,	//Register address
					Quantity	:=	1,	//Number of registers to be read
					pMemoryAddr	:=	ADR(fAct[i].FlowRel),		//Pointer to read data
					cbLength	:=	SIZEOF(fAct[i].FlowRel),	//Size of read data
					Timeout		:=	T#5S,				//Time to wait for the slave to respond
					Execute		:=	TRUE
				);
			ELSE
				fbModK8.ReadRegs(
					UnitID		:=	i,	//Modbus address of slave
					MBAddr		:=	6,	//Register address
					Quantity	:=	1,	//Number of registers to be read
					pMemoryAddr	:=	ADR(fAct[i].FlowRel),		//Pointer to read data
					cbLength	:=	SIZEOF(fAct[i].FlowRel),	//Size of read data
					Timeout		:=	T#5S,				//Time to wait for the slave to respond
					Execute		:=	TRUE
				);
			END_IF
			Step	:=	8;
			
		8:	//finish reading process
			IF (i=1) OR (i=3) OR (i=5) OR (i=7) THEN
				fbModK7.ReadRegs(Execute:=FALSE, Error=>bModErr, ErrorID=>ErrID);
				IF NOT fbModK7.BUSY THEN
					Step	:=	9;	//go to next step when reading process has finished
				END_IF
				IF fbModK7.Error THEN
					Step	:=	99;
				END_IF
			ELSE
				fbModK8.ReadRegs(Execute:=FALSE, Error=>bModErr, ErrorID=>ErrID);
				IF NOT fbModK8.BUSY THEN
					Step	:=	9;	//go to next step when reading process has finished
				END_IF
				IF fbModK8.Error THEN
					Step	:=	99;
				END_IF
			END_IF
	
		9:	//start reading absolute volume flow
			IF (i=1) OR (i=3) OR (i=5) OR (i=7) THEN
				fbModK7.ReadRegs(
					UnitID		:=	i,	//Modbus address of slave
					MBAddr		:=	7,	//Register address
					Quantity	:=	1,	//Number of registers to be read
					pMemoryAddr	:=	ADR(fAct[i].FlowAbs),		//Pointer to read data
					cbLength	:=	SIZEOF(fAct[i].FlowAbs),	//Size of read data
					Timeout		:=	T#5S,				//Time to wait for the slave to respond
					Execute		:=	TRUE
				);
			ELSE
				fbModK8.ReadRegs(
					UnitID		:=	i,	//Modbus address of slave
					MBAddr		:=	7,	//Register address
					Quantity	:=	1,	//Number of registers to be read
					pMemoryAddr	:=	ADR(fAct[i].FlowAbs),		//Pointer to read data
					cbLength	:=	SIZEOF(fAct[i].FlowAbs),	//Size of read data
					Timeout		:=	T#5S,				//Time to wait for the slave to respond
					Execute		:=	TRUE
				);
			END_IF
			Step	:=	10;
			
		10:	//finish reading process
			IF (i=1) OR (i=3) OR (i=5) OR (i=7) THEN
				fbModK7.ReadRegs(Execute:=FALSE, Error=>bModErr, ErrorID=>ErrID);
				IF NOT fbModK7.BUSY THEN
					Step	:=	11;	//go to next step when reading process has finished
				END_IF
				IF fbModK7.Error THEN
					Step	:=	99;
				END_IF
			ELSE
				fbModK8.ReadRegs(Execute:=FALSE, Error=>bModErr, ErrorID=>ErrID);
				IF NOT fbModK8.BUSY THEN
					Step	:=	11;	//go to next step when reading process has finished
				END_IF
				IF fbModK8.Error THEN
					Step	:=	99;
				END_IF
			END_IF	
				
		11:	//go to next nozzle or finish operation
			i	:=	i+1;
			IF i <= 10 THEN
				Step	:=	1;	//start process for next nozzle
			ELSE
				Step	:=	12;
			END_IF
			
		12:	//prepare next operation
			i		:=	1;
			Step	:=	1;
			
		20: //Control override
			nZwang	:=	2;
			IF (i=1) OR (i=3) OR (i=5) OR (i=7) THEN
					fbModK7.WriteSingleRegister(
						UnitID		:=	i,	//Modbus address of slave
						MBAddr		:=	1,	//Register address
						Quantity	:=	1,	//Number of registers to be written
						pMemoryAddr	:=	ADR(nZwang),		//Pointer to write data
						cbLength	:=	SIZEOF(nZwang),	//Size of write data
						Timeout		:=	T#5S,				//Time to wait for the slave to respond
						Execute		:=	TRUE
					);
				ELSE
					fbModK8.WriteSingleRegister(
						UnitID		:=	i,	//Modbus address of slave
						MBAddr		:=	1,	//Register address
						Quantity	:=	1,	//Number of registers to be written
						pMemoryAddr	:=	ADR(nZwang),		//Pointer to write data
						cbLength	:=	SIZEOF(nZwang),	//Size of write data
						Timeout		:=	T#5S,				//Time to wait for the slave to respond
						Execute		:=	TRUE
					);
				END_IF
				Step	:=	21;
		
			21:
			IF (i=1) OR (i=3) OR (i=5) OR (i=7) THEN
				fbModK7.WriteSingleRegister(Execute:=FALSE, Error=>bModErr, ErrorID=>ErrID);
				IF NOT fbModK7.BUSY THEN
					Step	:=	3;	//go to next step when writing process has finished
				END_IF
				IF fbModK7.Error THEN
					Step	:=	99;
				END_IF
			ELSE
				fbModK8.WriteSingleRegister(Execute:=FALSE, Error=>bModErr, ErrorID=>ErrID);
				IF NOT fbModK8.BUSY THEN
					Step	:=	3;	//go to next step when writing process has finished
				END_IF
				IF fbModK8.Error THEN
					Step	:=	99;
				END_IF
			END_IF
			
			30: //End control override
				nZwang	:=	0;
				IF (i=1) OR (i=3) OR (i=5) OR (i=7) THEN
					fbModK7.WriteSingleRegister(
						UnitID		:=	i,	//Modbus address of slave
						MBAddr		:=	1,	//Register address
						Quantity	:=	1,	//Number of registers to be written
						pMemoryAddr	:=	ADR(nZwang),		//Pointer to write data
						cbLength	:=	SIZEOF(nZwang),	//Size of write data
						Timeout		:=	T#5S,				//Time to wait for the slave to respond
						Execute		:=	TRUE
					);
				ELSE
					fbModK8.WriteSingleRegister(
						UnitID		:=	i,	//Modbus address of slave
						MBAddr		:=	1,	//Register address
						Quantity	:=	1,	//Number of registers to be written
						pMemoryAddr	:=	ADR(nZwang),		//Pointer to write data
						cbLength	:=	SIZEOF(nZwang),	//Size of write data
						Timeout		:=	T#5S,				//Time to wait for the slave to respond
						Execute		:=	TRUE
					);
				END_IF
				Step	:=	31;
		
			31:
			IF (i=1) OR (i=3) OR (i=5) OR (i=7) THEN
				fbModK7.WriteSingleRegister(Execute:=FALSE, Error=>bModErr, ErrorID=>ErrID);
				IF NOT fbModK7.BUSY THEN
					bZwang[i]	:=	FALSE;
					Step	:=	1;	//start normal writing process
				END_IF
				IF fbModK7.Error THEN
					Step	:=	99;
				END_IF
			ELSE
				fbModK8.WriteSingleRegister(Execute:=FALSE, Error=>bModErr, ErrorID=>ErrID);
				IF NOT fbModK8.BUSY THEN
					bZwang[i]	:=	FALSE;
					Step	:=	1;	//start normal writing process
				END_IF
				IF fbModK8.Error THEN
					Step	:=	99;
				END_IF
			END_IF
			
		99:	//Error
			
	END_CASE

END_IF

END_FUNCTION_BLOCK

// ---- POUs/Components/FC_CoolingCurve.TcPOU
FUNCTION FC_CoolingCurve : REAL
VAR_INPUT
	fTempAmb 	: REAL; 		//Ambient temerature
	fSlope 		: REAL := -1; 	//Slope of heatcurve
	fOffset 	: REAL := 18;	//In °C; off set at T_amb=T_room °C
	ftr			: REAL := 24;	//In °C; the set room temperature
END_VAR
VAR
END_VAR

IF fTempAmb < ftr THEN
	FC_CoolingCurve := foffset;
ELSE
	FC_CoolingCurve := fOffset - (fTempAmb - ftR);
END_IF

END_FUNCTION

// ---- POUs/Components/FC_MeanOfArray.TcPOU
FUNCTION FC_MeanOfArray : REAL
VAR_INPUT CONSTANT
	n 		: INT;
	aArray 	: ARRAY [1..n] OF REAL;
END_VAR
VAR
	i 		: INT;
	fTemp 	: REAL	:= 0;
END_VAR

FOR i := 1 TO n DO
	fTemp := fTemp + aArray[i];
END_FOR

FC_MeanOfArray := fTemp / n;

END_FUNCTION

// ---- POUs/Test/HeatSupplySystem_Test/FB_HSSController_Test.TcPOU
FUNCTION_BLOCK FB_HSSController_Test EXTENDS FB_TestSuite
VAR
	(*Sum : FB_Sum;
    Result : UINT;
    ExpectedSum : UINT := 4;*)

END_VAR

METHOD PID_Test1 : BOOL
VAR
	//Sum : FB_Sum;
    //Result : UINT;
    //ExpectedSum : UINT := 4;
END_VAR
//TEST('TwoPlusTwoEqualsFour');
 
//Sum(one := 2, two := 2, result => Result);
 
//AssertEquals(Expected := ExpectedSum,
//             Actual := Result,
//             Message := 'The calculation is not correct');
 
//TEST_FINISHED();
END_METHOD

END_FUNCTION_BLOCK
